# B&R Automation Studio project PLC code - cp (part 7)

#### BRSE_MB_Config.c
```c
/*! \file BRSE_MB_Config.c */

#include "BRSE_MB_Main.h"

BRSE_MB_ServerCfg_typ gBRSE_MB_Internal;

/*! \interface BRSE_MB_Alloc
	\brief Server: Function for allocating a modbus server unit.

	\param[in] 	Unit	Identity of the unit (0-255)
	\param[in]	MaxCoils	The maximum number of coils (references) used in this unit.
	\param[in]	MaxHoldingRegisters	The maximum number of holding registers used in this unit.
	\param[in] MaxDiscreteInputs	The maximum number of discrete inputs used in this unit.
	\param[in] MaxInputRegisters	The maximum number of input registers used in this unit.
	\param[out] Returns a pointer to the internal structure. Can be used for debug purposes.

*/
unsigned long BRSE_MB_Alloc(unsigned char Unit, unsigned short MaxCoils, unsigned short MaxHoldingRegisters, unsigned short MaxDiscreteInputs, unsigned short MaxInputRegisters)
{
	UINT status = 0;
	if (gBRSE_MB_Internal.Unit[Unit].pCoils || gBRSE_MB_Internal.Unit[Unit].pDiscreteInputs ||
		gBRSE_MB_Internal.Unit[Unit].pInputRegisters || gBRSE_MB_Internal.Unit[Unit].pHoldingRegisters)
		return BRSE_MB_ERR_UNIT_ALLOCATED; /* Unit can only be allocated once */

	memset(&gBRSE_MB_Internal.Unit[Unit], 0, sizeof(gBRSE_MB_Internal.Unit[Unit]));
	gBRSE_MB_Internal.Unit[Unit].MaxCoils = MaxCoils;
	gBRSE_MB_Internal.Unit[Unit].MaxDiscreteInputs = MaxDiscreteInputs;
	gBRSE_MB_Internal.Unit[Unit].MaxHoldingRegisters = MaxHoldingRegisters;
	gBRSE_MB_Internal.Unit[Unit].MaxInputRegisters = MaxInputRegisters;

	if (MaxCoils > 0)
	{
		status = TMP_alloc(MaxCoils*sizeof(UDINT) , (void **)&(gBRSE_MB_Internal.Unit[Unit].pCoils));
		if (status == 0)
			memset((void *)gBRSE_MB_Internal.Unit[Unit].pCoils, 0, MaxCoils*sizeof(UDINT));
		else
			ERRxwarning(status,(UDINT)gBRSE_MB_Internal.Unit[Unit].pCoils,(void *)"Coils: No memory!");
	}

	if (status != 0) /* reset unit */
	{
		memset(&gBRSE_MB_Internal.Unit[Unit], 0, sizeof(gBRSE_MB_Internal.Unit[Unit]));
		return status;
	}

	if (MaxDiscreteInputs > 0)
	{
		status = TMP_alloc(MaxDiscreteInputs*sizeof(UDINT) , (void **)&(gBRSE_MB_Internal.Unit[Unit].pDiscreteInputs));
		if (status == 0)
			memset((void *)gBRSE_MB_Internal.Unit[Unit].pDiscreteInputs, 0, MaxDiscreteInputs*sizeof(UDINT));
		else
			ERRxwarning(status,(UDINT)gBRSE_MB_Internal.Unit[Unit].pDiscreteInputs,(void *)"DiscreteI: No memory!");
	}

	if (status != 0) /* reset unit */
	{
		memset(&gBRSE_MB_Internal.Unit[Unit], 0, sizeof(gBRSE_MB_Internal.Unit[Unit]));
		return status;
	}

	if (MaxHoldingRegisters > 0)
	{
		status = TMP_alloc(MaxHoldingRegisters*sizeof(UDINT) , (void **)&(gBRSE_MB_Internal.Unit[Unit].pHoldingRegisters));
		if (status == 0)
			memset((void *)gBRSE_MB_Internal.Unit[Unit].pHoldingRegisters, 0, MaxHoldingRegisters*sizeof(UDINT));
		else
			ERRxwarning(status,(UDINT)gBRSE_MB_Internal.Unit[Unit].pHoldingRegisters,(void *)"HoldingR: No memory!");
	}

	if (status != 0) /* reset unit */
	{
		memset(&gBRSE_MB_Internal.Unit[Unit], 0, sizeof(gBRSE_MB_Internal.Unit[Unit]));
		return status;
	}

	if (MaxInputRegisters > 0)
	{
		status = TMP_alloc(MaxInputRegisters*sizeof(UDINT) , (void **)&(gBRSE_MB_Internal.Unit[Unit].pInputRegisters));
		if (status == 0)
			memset((void *)gBRSE_MB_Internal.Unit[Unit].pInputRegisters, 0, MaxInputRegisters*sizeof(UDINT));
		else
			ERRxwarning(status,(UDINT)gBRSE_MB_Internal.Unit[Unit].pInputRegisters,(void *)"InputReg:  No memory!");
	}

	if (status != 0) /* reset unit */
	{
		memset(&gBRSE_MB_Internal.Unit[Unit], 0, sizeof(gBRSE_MB_Internal.Unit[Unit]));
	}

	return (unsigned long)&gBRSE_MB_Internal;
}

/*! \interface BRSE_MB_Coil
	\brief Server: Function binding a coil to a variable

	Note that this function uses relative modbus adressing. Reference 0 corresponds to Modbus adress 1.

	\param[in] 	Unit	Identity of the unit (0-255)
	\param[in]	Reference	Coil address within unit (0..MaxCoils-1 in Alloc)
	\param[in]	VariableAddress	Address of the boolean variable.
	\param[out] Returns 0 or an error code.
*/
unsigned short BRSE_MB_Coil(unsigned char Unit, unsigned short Reference, unsigned long PvAddress)
{
	UDINT *coils;
	if (Reference >= gBRSE_MB_Internal.Unit[Unit].MaxCoils || PvAddress == 0)
		return BRSE_MB_ERR_REFERENCE;
	coils = (UDINT *)gBRSE_MB_Internal.Unit[Unit].pCoils; /* use as dynamic UDINT[] */
	coils[Reference] = PvAddress;
	return 0;
}

/*! \interface BRSE_MB_HoldingRegister
	\brief Server: Function binding a holding register to a variable

	Note that this function uses relative modbus adressing. Reference 0 corresponds to Modbus adress 40001.

	\param[in] 	Unit	Identity of the unit (0-255)
	\param[in]	Reference	Holding register address within unit (0..MaxHoldingRegisters-1 in Alloc)
	\param[in]	VariableAddress	Address of the integer variable.
	\param[out] Returns 0 or an error code.
*/
unsigned short BRSE_MB_HoldingRegister(unsigned char Unit, unsigned short Reference, unsigned long PvAddress)
{
	UDINT *holdingRegisters;
	if (Reference >= gBRSE_MB_Internal.Unit[Unit].MaxHoldingRegisters || PvAddress == 0)
		return BRSE_MB_ERR_REFERENCE;
	holdingRegisters = (UDINT *)gBRSE_MB_Internal.Unit[Unit].pHoldingRegisters; /* use as dynamic UDINT[] */
	holdingRegisters[Reference] = PvAddress;
	return 0;
}

/*! \interface BRSE_MB_4ByteHoldingRegister
	\brief Server: Function binding a 4 byte variable to 2 holding registers

	Note that this function uses relative modbus adressing. Reference 0 corresponds to Modbus adress 40001.

	\param[in] 	Unit	Identity of the unit (0-255)
	\param[in]	Reference	Holding register address within unit (0..MaxHoldingRegisters-1 in Alloc). Next free modbus address will be Reference+2 as the function assumes that you bind a 4-byte variable.
	\param[in]	VariableAddress	Address of the 4 byte variable.
	\param[out] Returns 0 or an error code.
*/
unsigned short BRSE_MB_4ByteHoldingRegister(unsigned char Unit, unsigned short Reference, unsigned long PvAddress)
{
	UDINT *holdingRegisters;
	if (Reference + 1 >= gBRSE_MB_Internal.Unit[Unit].MaxHoldingRegisters || PvAddress == 0)
		return BRSE_MB_ERR_REFERENCE;
	holdingRegisters = (UDINT *)gBRSE_MB_Internal.Unit[Unit].pHoldingRegisters; /* use as dynamic UDINT[] */
	holdingRegisters[Reference] = 1;
	holdingRegisters[Reference + 1] = PvAddress;
	return 0;
}
/*! \interface BRSE_MB_InputRegister
	\brief Server: Function binding a input register to a variable

	Note that this function uses relative modbus adressing. Reference 0 corresponds to Modbus adress 30001

	\param[in] 	Unit	Identity of the unit (0-255)
	\param[in]	Reference	Input register address within unit (0..MaxInputRegister-1 in Alloc)
	\param[in]	VariableAddress	Address of the integer variable.
	\param[out] Returns 0 or an error code.
*/
unsigned short BRSE_MB_InputRegister(unsigned char Unit, unsigned short Reference, unsigned long PvAddress)
{
	UDINT *inputRegisters;
	if (Reference >= gBRSE_MB_Internal.Unit[Unit].MaxInputRegisters || PvAddress == 0)
		return BRSE_MB_ERR_REFERENCE;
	inputRegisters = (UDINT *)gBRSE_MB_Internal.Unit[Unit].pInputRegisters; /* use as dynamic UDINT[] */
	inputRegisters[Reference] = PvAddress;
	return 0;
}

/*! \interface BRSE_MB_DiscreteInput
	\brief Server: Function binding a coil to a variable

	Note that this function uses relative modbus adressing. Reference 0 corresponds to Modbus adress 10001.

	\param[in] 	Unit	Identity of the unit (0-255)
	\param[in]	Reference	Coil address within unit (0..MaxDiscreteInputs-1 in Alloc)
	\param[in]	VariableAddress	Address of the boolean variable.
	\param[out] Returns 0 or an error code.
*/
unsigned short BRSE_MB_DiscreteInput(unsigned char Unit, unsigned short Reference, unsigned long PvAddress)
{
	UDINT *discreteInputs;
	if (Reference >= gBRSE_MB_Internal.Unit[Unit].MaxDiscreteInputs || PvAddress == 0)
		return BRSE_MB_ERR_REFERENCE;
	discreteInputs = (UDINT *)gBRSE_MB_Internal.Unit[Unit].pDiscreteInputs; /* use as dynamic UDINT[] */
	discreteInputs[Reference] = PvAddress;
	return 0;
}
```

#### BRSE_MB_Server.c
```c
/*! \file BRSE_MB_Server.c */

#include <bur/plctypes.h>
#include "BRSE_MB.h"
#include "BRSE_MB_Main.h"

/***************************/
/* Necessary byte swapping */
/***************************/
#ifdef _SG4
	#define SWAPUINT	swapUINT
	#define SWAPINT		swapINT
#else
	#define SWAPUINT
	#define SWAPINT
#endif

extern BRSE_MB_ServerCfg_typ gBRSE_MB_Internal; /* declared in BRSE_MB_Config.c */

 /*!
	\interface BRSE_MB_Server
	\brief Server: Interprets a byte buffer and creates a response to it according to modbus specification.
	Units and variables are configured with other BRSE_MB-functions.

	\param[in] Unit			The unit identifier (0-254)
	\param[in]	ClientFormat	Set the format of 4 byte variables to Intel or Motorola. BRSE_MB_INTEL / BRSE_MB_MOTOROLA

	\param[in] InputBuffer	The modbus byte buffer to respond to.
		Byte 0 is the function code.
		Byte 1-2 is the reference number (offset within unit where to start reading/writing).

	\param[out] OutputBuffer	The response buffer
	\param[out] BufferLength	The total number of bytes in the output buffer
	\param[out] Status			Return status.

*/
void BRSE_MB_Server(struct BRSE_MB_Server* inst)
{
	UINT	uintVar;
	/*****************************************/
	/* Check inputs and reset function block */
	/*****************************************/
	if (
		 (	!gBRSE_MB_Internal.Unit[inst->Unit].pCoils && !gBRSE_MB_Internal.Unit[inst->Unit].pDiscreteInputs &&
			!gBRSE_MB_Internal.Unit[inst->Unit].pInputRegisters && !gBRSE_MB_Internal.Unit[inst->Unit].pHoldingRegisters)
		)/* Unit not allocated */
	{
		inst->Status = BRSE_MB_ERR_ILLEGAL_FUNCTION; /* Unit is unconfigured and cannot process any request */
		return;
	}

	memset(&inst->OutputBuffer, 0, sizeof(inst->OutputBuffer));
	memset(&inst->Request, 0, sizeof(inst->Request));

	/*****************************/
	/* Parse request information */
	/*****************************/

	/* Function code (byte 0) */
	inst->Request.Type = inst->InputBuffer[0];
	if (inst->Request.Type == 0) /* FC 0 does not exist */
	{
		inst->Status = BRSE_MB_ERR_ILLEGAL_FUNCTION;
		return;
	}
	/* Reference number (byte 1,2) */
	memcpy(&uintVar, &inst->InputBuffer[1], sizeof(uintVar));
	inst->Request.StartAddr = SWAPUINT(uintVar);

	if(inst->Request.Type == BRSE_MB_WRITE_SINGLE_COIL || inst->Request.Type == BRSE_MB_WRITE_SINGLE_REGISTER)
	{
		inst->Request.Quantity = 1;
	}
	else /* Word/bit count (byte 3,4) */
	{
		memcpy(&uintVar, &inst->InputBuffer[3], sizeof(uintVar));
		inst->Request.Quantity = SWAPUINT(uintVar);
	}
	if (inst->Request.Quantity == 0)
	{
		inst->Status = BRSE_MB_ERR_ILLEGAL_DATA_ADDRESS;
		return;
	}

	/**************************************/
	/* Analyze request and build response */
	/**************************************/
	inst->OutputBuffer[0] = inst->Request.Type; /* Echo function code */

	switch(inst->Request.Type)
	{
		case BRSE_MB_READ_COILS:					/* 0x01 */
			inst->Status = BRSE_MB_ReadCoils(inst);
			break;

		case BRSE_MB_READ_DISCRETE_INPUTS:			/* 0x02 */
			inst->Status = BRSE_MB_ReadDiscreteInputs(inst);
			break;

		case BRSE_MB_READ_HOLDING_REGISTERS:		/* 0x03 */
			inst->Status = BRSE_MB_ReadHoldingRegisters(inst);
			break;

		case BRSE_MB_READ_INPUT_REGISTERS:			/* 0x04 */
			inst->Status = BRSE_MB_ReadInputRegisters(inst);
			break;

		case BRSE_MB_WRITE_SINGLE_COIL:				/* 0x05 */
			inst->Status = BRSE_MB_WriteSingleCoil(inst);
			break;

		case BRSE_MB_WRITE_SINGLE_REGISTER:			/* 0x06 */
			inst->Status = BRSE_MB_WriteSingleRegister(inst);
			break;

		case BRSE_MB_WRITE_MULTIPLE_COILS:			/* 0x0F */
			inst->Status = BRSE_MB_WriteMultipleCoils(inst);
			break;

		case BRSE_MB_WRITE_MULTIPLE_REGISTERS:		/* 0x10 */
			inst->Status = BRSE_MB_WriteMultipleRegisters(inst);
			break;

		default:
			inst->Status = BRSE_MB_ERR_ILLEGAL_FUNCTION;
			break;
	}
	if (inst->Status != 0) /* Reset outputs */
		memset(&inst->OutputBuffer, 0, sizeof(inst->OutputBuffer));

}

UINT BRSE_MB_ReadCoils(struct BRSE_MB_Server* inst)
{
	UDINT 				*coils;
	if(inst->Request.StartAddr + inst->Request.Quantity <= gBRSE_MB_Internal.Unit[inst->Unit].MaxCoils
		&& inst->Request.Quantity <= BRSE_MB_MAX_COILS
		&& gBRSE_MB_Internal.Unit[inst->Unit].pCoils)
	{
		coils = (UDINT *)gBRSE_MB_Internal.Unit[inst->Unit].pCoils; /* use as dynamic UDINT[] */
		return BRSE_MB_FillDigitalBuffer(inst, coils);
	}
	else
	{
		return BRSE_MB_ERR_ILLEGAL_DATA_ADDRESS;
	}
}

UINT BRSE_MB_ReadDiscreteInputs(struct BRSE_MB_Server* inst)
{
	UDINT 				*discreteInputs;
	if(inst->Request.StartAddr + inst->Request.Quantity <= gBRSE_MB_Internal.Unit[inst->Unit].MaxDiscreteInputs
		&& inst->Request.Quantity <= BRSE_MB_MAX_DISCRETE_INPUTS
		&& gBRSE_MB_Internal.Unit[inst->Unit].pDiscreteInputs)
	{
		discreteInputs = (UDINT *)gBRSE_MB_Internal.Unit[inst->Unit].pDiscreteInputs; /* use as dynamic UDINT[] */
		return BRSE_MB_FillDigitalBuffer(inst, discreteInputs);
	}
	else
	{
		return BRSE_MB_ERR_ILLEGAL_DATA_ADDRESS;
	}
}

UINT BRSE_MB_ReadHoldingRegisters(struct BRSE_MB_Server* inst)
{
	UDINT *holdingRegisters;
	if (inst->Request.StartAddr + inst->Request.Quantity <= gBRSE_MB_Internal.Unit[inst->Unit].MaxHoldingRegisters
		&& inst->Request.Quantity <= BRSE_MB_MAX_HOLDING_REG_READ
		&& gBRSE_MB_Internal.Unit[inst->Unit].pHoldingRegisters)
	{
		holdingRegisters = (UDINT *)gBRSE_MB_Internal.Unit[inst->Unit].pHoldingRegisters; /* use as dynamic UDINT[] */
		return BRSE_MB_FillRegisterBuffer(inst, holdingRegisters);
	}
	else
	{
		return BRSE_MB_ERR_ILLEGAL_DATA_ADDRESS;
	}
}

UINT BRSE_MB_ReadInputRegisters(struct BRSE_MB_Server* inst)
{
	UDINT *inputRegisters;
	if (inst->Request.StartAddr + inst->Request.Quantity <= gBRSE_MB_Internal.Unit[inst->Unit].MaxInputRegisters
		&& inst->Request.Quantity <= BRSE_MB_MAX_INPUT_REG_READ
		&& gBRSE_MB_Internal.Unit[inst->Unit].pInputRegisters)
	{
		inputRegisters = (UDINT *)gBRSE_MB_Internal.Unit[inst->Unit].pInputRegisters; /* use as dynamic UDINT[] */
		return BRSE_MB_FillRegisterBuffer(inst, inputRegisters);
	}
	else
	{
		return BRSE_MB_ERR_ILLEGAL_DATA_ADDRESS;
	}
}

/*
 Response looks like
   Byte
	0:			FC
	1-2:		Reference
	3:			FF=0N, 00=OFF
	4:			0

	sets BufferLength = 5
 */
UINT BRSE_MB_WriteSingleCoil(struct BRSE_MB_Server* inst)
{
	UINT uintVar;
	UINT value;
	UDINT *coils;

	inst->BufferLength = 5;
	if(inst->Request.StartAddr < gBRSE_MB_Internal.Unit[inst->Unit].MaxCoils && gBRSE_MB_Internal.Unit[inst->Unit].pCoils)
	{
		coils = (UDINT *)gBRSE_MB_Internal.Unit[inst->Unit].pCoils; /* use as dynamic UDINT[] */
		memcpy(&uintVar, &inst->InputBuffer[3], sizeof(uintVar)); /* value */
		value = SWAPUINT(uintVar);

		memcpy(&inst->OutputBuffer[1], &inst->InputBuffer[1], 2); /* Reference: 2 byte */
		memcpy(&inst->OutputBuffer[3], &inst->InputBuffer[3], 2); /* Value: 2 byte */

		if (coils[inst->Request.StartAddr])
		{
			if(value == BRSE_MB_ON)
				*((BOOL*)(coils[inst->Request.StartAddr])) = 1;
			else
				*((BOOL*)(coils[inst->Request.StartAddr])) = 0;
		}
	}
	else
	{
		return BRSE_MB_ERR_ILLEGAL_DATA_ADDRESS;
	}
	return 0;
}

/*
 Response looks like
   Byte
	0:			FC
	1-2:		Reference
	3-4:		Register value

	sets BufferLength = 5
 */
UINT BRSE_MB_WriteSingleRegister(struct BRSE_MB_Server* inst)
{
	INT intVar;
	INT value;
	UDINT *holdingRegisters;

	inst->BufferLength = 5;

	if(inst->Request.StartAddr < gBRSE_MB_Internal.Unit[inst->Unit].MaxHoldingRegisters && gBRSE_MB_Internal.Unit[inst->Unit].pHoldingRegisters)
	{
		holdingRegisters = (UDINT *)gBRSE_MB_Internal.Unit[inst->Unit].pHoldingRegisters; /* use as dynamic UDINT[] */
		memcpy(&intVar, &(inst->InputBuffer[3]), sizeof(intVar)); /* value */
		value = SWAPUINT(intVar);

		memcpy(&inst->OutputBuffer[1], &inst->InputBuffer[1], 2); /* Reference: 2 byte */
		memcpy(&inst->OutputBuffer[3], &inst->InputBuffer[3], 2); /* Value: 2 byte */

		if (holdingRegisters[inst->Request.StartAddr] > 1) /*check that its not a 4-byte holding!*/
			*((INT*)(holdingRegisters[inst->Request.StartAddr])) = value;
		else
			return BRSE_MB_ERR_ILLEGAL_DATA_ADDRESS;
	}
	else
	{
		return BRSE_MB_ERR_ILLEGAL_DATA_ADDRESS;
	}

	return 0;
}

/*
 Response looks like
   Byte
	0:			FC
	1-2:		Reference
	3-4:		Bit count

	sets BufferLength = 5
 */
UINT BRSE_MB_WriteMultipleCoils(struct BRSE_MB_Server* inst)
{
	UINT i;
	UDINT *coils;

	inst->BufferLength = 5;
	if(inst->Request.StartAddr + inst->Request.Quantity <= gBRSE_MB_Internal.Unit[inst->Unit].MaxCoils
		&& inst->Request.Quantity <= BRSE_MB_MAX_COILS_WRITE
		&& gBRSE_MB_Internal.Unit[inst->Unit].pCoils)
	{
		coils = (UDINT *)gBRSE_MB_Internal.Unit[inst->Unit].pCoils; /* use as dynamic UDINT[] */
		memcpy(&inst->OutputBuffer[1], &inst->InputBuffer[1], 2);		/* Reference: 2 byte */
		memcpy(&inst->OutputBuffer[3], &inst->InputBuffer[3], 2);  	/* Bit count: 2 byte */

		for(i=0; i < inst->Request.Quantity; i++)
		{
			if (coils[inst->Request.StartAddr+i])
			{
				if ((inst->InputBuffer[6 + (i/8)] & (USINT)(0x01 << (i%8))) && (coils[inst->Request.StartAddr+i]))
					*((BOOL*)(coils[inst->Request.StartAddr+i])) = 1;
				else
					*((BOOL*)(coils[inst->Request.StartAddr+i])) = 0;
			}
		}
		return 0;
	}
	else
	{
		return BRSE_MB_ERR_ILLEGAL_DATA_ADDRESS;
	}

}
/*
 Response looks like
   Byte
	0:			FC
	1-2:		Reference
	3-4:		Word count

	sets BufferLength = 5
 */
UINT BRSE_MB_WriteMultipleRegisters(struct BRSE_MB_Server* inst)
{
	INT							int_var1, int_var2;
	UINT						i;
	UDINT *holdingRegisters;

	inst->BufferLength = 5;

	if (inst->Request.StartAddr + inst->Request.Quantity <= gBRSE_MB_Internal.Unit[inst->Unit].MaxHoldingRegisters
		&& inst->Request.Quantity <= BRSE_MB_MAX_HOLDING_REG_WRITE
		&& gBRSE_MB_Internal.Unit[inst->Unit].pHoldingRegisters)
	{

			holdingRegisters = (UDINT *)gBRSE_MB_Internal.Unit[inst->Unit].pHoldingRegisters; /* use as dynamic UDINT[] */
			memcpy(&inst->OutputBuffer[1], &inst->InputBuffer[1], 2);	/* 	Reference: 2 byte */
			memcpy(&inst->OutputBuffer[3], &inst->InputBuffer[3], 2); 	/* Value: 2 byte */

			for(i=0; i < inst->Request.Quantity; i++)
			{
				if (holdingRegisters[inst->Request.StartAddr+i] == 0)
				{
					return BRSE_MB_ERR_ILLEGAL_DATA_ADDRESS;
				}

				if (holdingRegisters[inst->Request.StartAddr+i] == 1 && holdingRegisters[inst->Request.StartAddr+i+1]) /* 4 byte variable */
				{
					memcpy(&int_var1, &inst->InputBuffer[6+(i*2)], sizeof(int_var1));
					memcpy(&int_var2, &inst->InputBuffer[6+(i*2)+2], sizeof(int_var2));
					if (inst->ClientFormat == BRSE_MB_INTEL )
					{
						#ifdef _SG4
						*((INT*)(holdingRegisters[inst->Request.StartAddr+i+1])) = SWAPINT(int_var1);
						*((INT*)(holdingRegisters[inst->Request.StartAddr+i+1]+2)) = SWAPINT(int_var2);
						#else
						*((INT*)(holdingRegisters[inst->Request.StartAddr+i+1])) = SWAPINT(int_var2);
						*((INT*)(holdingRegisters[inst->Request.StartAddr+i+1]+2)) = SWAPINT(int_var1);
						#endif
					}
					else
					{
						#ifdef _SG4
						*((INT*)(holdingRegisters[inst->Request.StartAddr+i+1])) = SWAPINT(int_var2);
						*((INT*)(holdingRegisters[inst->Request.StartAddr+i+1]+2)) = SWAPINT(int_var1);
						#else
						*((INT*)(holdingRegisters[inst->Request.StartAddr+i+1])) = SWAPINT(int_var1);
						*((INT*)(holdingRegisters[inst->Request.StartAddr+i+1]+2)) = SWAPINT(int_var2);
						#endif
					}

					i++;
				}
				else if (holdingRegisters[inst->Request.StartAddr+i] > 1) /* Normal 2 byte register */
				{
					memcpy(&int_var1, &inst->InputBuffer[6+(i*2)], sizeof(int_var1));
					*((INT*)(holdingRegisters[inst->Request.StartAddr+i])) = SWAPINT(int_var1);
				}
			}

			return 0;
	}
	else
	{
		return BRSE_MB_ERR_ILLEGAL_DATA_ADDRESS;
	}
}

/*********************/
/* Utility functions */
/*********************/
/*
 Response looks like
   Byte
	0:			FC
	1:			Byte count of response (B=(bit count +7)/8)
	2-(B+1):	Bit values

	sets BufferLength = 2+B
 */
UINT BRSE_MB_FillDigitalBuffer(struct BRSE_MB_Server* inst, UDINT *boolPtrArray)
{
	UINT				i;
	USINT				byte_nr;
	/* Number of bytes in response (1) */
	if ((inst->Request.Quantity % 8) > 0)	byte_nr = (inst->Request.Quantity / 8) + 1;
	else									byte_nr = (inst->Request.Quantity / 8);
	inst->OutputBuffer[1] = byte_nr;

	/* Value of boolean boolPtrArray (2->byte_nr) */
	for(i = 0; i < inst->Request.Quantity; i++)
	{
		/* if pv assigned and true */
		if( boolPtrArray[inst->Request.StartAddr+i] && (*((BOOL *)boolPtrArray[inst->Request.StartAddr+i])))
			inst->OutputBuffer[2 + (i/8)] = inst->OutputBuffer[2 + (i/8)] | (USINT)(0x01 << (i%8));
		else
			inst->OutputBuffer[2 + (i/8)] = inst->OutputBuffer[2 + (i/8)] & (USINT)~(0x01 << (i%8));

	}
	inst->BufferLength = 2+byte_nr;
	return 0;
}

/*
 Response looks like
   Byte
	0:			FC
	1:			Byte count of response (B=2*word count)
	2-(B+1):	Register values (1-125)

	returns BufferLength = 2+2*(word count)
 */
UINT BRSE_MB_FillRegisterBuffer(struct BRSE_MB_Server* inst, UDINT *intPtrArray)
{
	INT				int_var1, int_var2;
	UINT			i;

	inst->OutputBuffer[1] = inst->Request.Quantity * 2; /* nbr data bytes */

	for(i = 0; i < inst->Request.Quantity; i++)
	{
		if(intPtrArray[inst->Request.StartAddr + i])
		{
			if(intPtrArray[inst->Request.StartAddr + i] == 1 && intPtrArray[inst->Request.StartAddr + i + 1]) /*4-byte*/
			{
				int_var1 = SWAPINT(*((INT*)(intPtrArray[inst->Request.StartAddr + i + 1])));
				int_var2 = SWAPINT(*((INT*)(intPtrArray[inst->Request.StartAddr + i + 1]+2)));

				if(inst->ClientFormat == BRSE_MB_INTEL)
				{
					#ifdef _SG4
						memcpy(&inst->OutputBuffer[2 + (i*2)], &int_var1, sizeof(int_var1));
						memcpy(&inst->OutputBuffer[2 + ((i+1)*2)], &int_var2, sizeof(int_var2));
					#else
						memcpy(&inst->OutputBuffer[2 + (i*2)], &int_var2, sizeof(int_var2));
						memcpy(&inst->OutputBuffer[2 + ((i+1)*2)], &int_var1, sizeof(int_var1));
					#endif
				}
				else
				{
					#ifdef _SG4
						memcpy(&inst->OutputBuffer[2 + (i*2)], &int_var2, sizeof(int_var2));
						memcpy(&inst->OutputBuffer[2 + ((i+1)*2)], &int_var1, sizeof(int_var1));
					#else
						memcpy(&inst->OutputBuffer[2 + (i*2)], &int_var1, sizeof(int_var1));
						memcpy(&inst->OutputBuffer[2 + ((i+1)*2)], &int_var2, sizeof(int_var2));
					#endif
				}

				i++;
			}
			else if(intPtrArray[inst->Request.StartAddr + i] > 1) /*just in case, normally it shouldnt be 1 here anyhow*/
			{
				int_var1 = SWAPINT(*((INT*)(intPtrArray[inst->Request.StartAddr + i])));
				memcpy(&inst->OutputBuffer[2 + (i*2)], &int_var1, sizeof(int_var1));
			}
		}
		else /*bad pointer*/
		{
			int_var1 = 0;
			memcpy(&inst->OutputBuffer[2 + (i*2)], &int_var1, sizeof(int_var1));
		}
	}
	inst->BufferLength = 2+2*inst->Request.Quantity;
	return 0;
}
```

#### MB_RequestQueue.c
```c
/*! \file MB_RequestQueue.c */

#include <bur/plctypes.h>
#include "BRSE_MB.h"
#include "BRSE_MB_Main.h"

#define	BUSY				65535

extern MB_ClientStruct_typ gMB_ClientInternal;

UINT MB_AckClientRequest(USINT ClientID, UINT ReturnStatus)
{
	MB_Client_typ *pQueue;
	MB_ClientQueueItem_typ *pQueueItem;
	UINT status = 0;

	if (gMB_ClientInternal.pClients[ClientID] == 0)
		return MB_ERR_CLIENT_NOT_ALLOCATED;

	pQueue = (MB_Client_typ *)gMB_ClientInternal.pClients[ClientID];
	if ((*pQueue).Lock)
	{
		status = BUSY;
		return status;
	}

	/* -- Begin synchronized block -- */
	(*pQueue).Lock = 1; /* prevent others from reading from / writing to queue */
	pQueueItem = &((*pQueue).Queue[(*pQueue).IndexExec]);
	(*((UINT *) ((*pQueueItem).StatusAddr))) = ReturnStatus;
	(*pQueue).IndexExec++;
	(*pQueue).IndexExec %= (MB_QUEUE_SIZE+1);
	memset(pQueueItem, 0, sizeof(*pQueueItem));
	(*pQueue).Lock = 0;
	/* -- End synchronized block -- */
	return status;
}

UINT MB_AddToRequestQueue(USINT clientID, USINT fc, UINT quantity, UINT startAddress, UDINT variableAddress, UDINT statusAddress, USINT Unit)
{
	MB_Client_typ *pQueue;
	MB_ClientQueueItem_typ *pQueueItem;
	UINT status = 0;

	if (gMB_ClientInternal.pClients[clientID] == 0)
		return MB_ERR_CLIENT_NOT_ALLOCATED;

	pQueue = (MB_Client_typ *)gMB_ClientInternal.pClients[clientID];
	if ((*pQueue).Lock)
	{
		status = BUSY;
		return status;
	}

	/* -- Begin synchronized block -- */
	(*pQueue).Lock = 1; /* prevent others from reading from / writing to queue */
	pQueueItem = &((*pQueue).Queue[(*pQueue).IndexInsert]);
	if (((*pQueue).IndexExec == (*pQueue).IndexInsert) && ((*pQueueItem).VariableAddr != 0))
	{
		status = MB_ERR_QUEUE_FULL;
	}
	else
	{
		(*((UINT *)statusAddress)) = BUSY;
		(*pQueueItem).Request.Unit = Unit;
		(*pQueueItem).Request.Quantity = quantity;
		(*pQueueItem).Request.Type = fc;
		(*pQueueItem).Request.StartAddr = startAddress;
		(*pQueueItem).VariableAddr = variableAddress;
		(*pQueueItem).StatusAddr = statusAddress;
		(*pQueue).IndexInsert++;
		(*pQueue).IndexInsert %= (MB_QUEUE_SIZE+1);
	}
	(*pQueue).Lock = 0;
	/* -- End synchronized block -- */
	return status;
}

USINT MB_QueueStatus(USINT ClientID)
{
	MB_Client_typ *pQueue;
	USINT status = 0;

	if (gMB_ClientInternal.pClients[ClientID] == 0)
		return 0;

	pQueue = (MB_Client_typ *)gMB_ClientInternal.pClients[ClientID];
	if ((*pQueue).Lock)
	{
		return 1;
	}
	/* Synchronized block */
	(*pQueue).Lock = 1;
	if ((*pQueue).IndexExec == (*pQueue).IndexInsert) /* queue empty */
		status = 0;
	else
		status = 1;
	(*pQueue).Lock = 0;
	/* Synchronized end */
	return status;
}
```

### Library Logical/ExtPack/_Comms/ModbusComms/ModbusComms_v1/Libraries/BRSE_MBT

#### BRSE_MBT.var
```iecst
VAR CONSTANT
	BRSE_MBT_MAX_BUFFER : UINT := 261;
	BRSE_MBT_MAX_CLIENT : USINT := 20;
	BRSE_MBT_ERR_TOO_MANY_CLIENTS : UINT := 30001;
	BRSE_MBT_LOG_MAX : UINT := 50;
	MBT_RECEIVE_TIMEOUT : UDINT := 3000; (*Await response timeout, ms (cycle time=0 --> never timeout)*)
	BRSE_MBT_RESEND_LIMIT : UINT := 5; (*Number of times to resend before trying to re-establish connection*)
	BRSE_MBT_RETRY_PERIOD : UINT := 10000; (*If error occurs on TcpOpen or TcpClient, wait this time before retrying. (cycle time assumed 10ms if set to 0)*)
	BRSE_DISCONNECT_TIMEOUT : TIME := T#60S; (*Disconnects clients after this time without activity*)
END_VAR
```

#### BRSE_MBT.fun
```iecst
FUNCTION_BLOCK BRSE_MBT_Server
	VAR_INPUT
		Enable : BOOL; (*Add your parameter comment*)
		ClientFormat : USINT;
		Port : UINT;
		SocketTimeout : UDINT; (*Linger time for incoming sockets*)
	END_VAR
	VAR_OUTPUT
		Status : UINT;
	END_VAR
	VAR
		FB_TcpOpen : TcpOpen;
		FB_TcpServer : TcpServer;
		FB_TcpCloseOld : TcpClose;
		FB_TcpCloseServer : TcpClose;
		FB_TcpClose : ARRAY[0..BRSE_MBT_MAX_CLIENT] OF TcpClose;
		Clients : ARRAY[0..BRSE_MBT_MAX_CLIENT] OF BRSE_MBT_Client_typ;
		Step : UINT;
		ClientNr : USINT;
		FB_BRSE_MB_Server : BRSE_MB_Server;
		Log : ARRAY[0..BRSE_MBT_LOG_MAX] OF STRING[100];
		LogIndex : UINT;
		TmpUINT : UINT;
		NewClient : BRSE_MBT_NewClient_typ;
		Error : UINT; (*Indicator to leave state when all fubs are done*)
		IsBusy : UINT; (*Indicates that one or more fubs are not ready to leave state*)
		TmpStr : STRING[10];
		LingerOptions : tcpLINGER_typ;
	END_VAR
END_FUNCTION_BLOCK

FUNCTION MBT_GetServerInternalStructAddr : UDINT (*Returns the allocated server struct address, i.e. a pointer to a BRSE_MBT_Internal_typ. Used only for debug purposes.*)
END_FUNCTION

FUNCTION MBT_GetClientInternalStructAddr : UDINT (*Returns the allocated client internal struct address, i.e. a pointer to a MBT_ClientInternal_typ. Used only for debug purposes.*)
END_FUNCTION

FUNCTION_BLOCK MBT_ServerExit (*Closes any open tcp port.*)
	VAR_OUTPUT
		Status : UINT;
	END_VAR
	VAR
		FB_TcpClose : TcpClose;
	END_VAR
END_FUNCTION_BLOCK

FUNCTION_BLOCK MBT_Client
	VAR_INPUT
		Enable : BOOL;
		ServerFormat : USINT;
		ClientID : USINT;
		IpAddr : STRING[18];
		Port : UINT;
		ConnectionTimeout : UDINT; (*Time in ms the client waits for new requests (from queue) before closing down the socket connection*)
		SocketTimeout : UDINT; (*Linger time for outgoing sockets*)
	END_VAR
	VAR_OUTPUT
		Status : UINT;
	END_VAR
	VAR
		Step : UINT;
		FB_MB_CreateClientRequest : MB_CreateClientRequest;
		FB_MB_PutClientResponse : MB_PutClientResponse;
		FB_TcpOpen : TcpOpen;
		FB_TcpClient : TcpClient;
		FB_TcpSend : TcpSend;
		FB_TcpRecive : TcpRecv;
		FB_TcpClose : TcpClose;
		FB_RTInfo : RTInfo;
		FB_TcpIoctl : TcpIoctl;
		RecvLen : UINT;
		SendBuffer : ARRAY[0..BRSE_MBT_MAX_BUFFER] OF USINT;
		ReceiveBuffer : ARRAY[0..BRSE_MBT_MAX_BUFFER] OF USINT;
		TransactionId : UINT;
		Timeout : UDINT;
		RecvTransactionId : UINT;
		ErrorStatus : UINT;
		ResendCounter : UINT;
		CycleTimeMs : UDINT; (*Task cycle time in ms*)
		ElapsedTime : UDINT;
		LingerOptions : tcpLINGER_typ;
	END_VAR
END_FUNCTION_BLOCK

FUNCTION_BLOCK MBT_ExitClient (*Closes any open tcp port.*)
	VAR_INPUT
		ClientID : USINT; (*Add your parameter comment*)
	END_VAR
	VAR_OUTPUT
		Status : UINT;
	END_VAR
	VAR
		FB_TcpClose : TcpClose;
	END_VAR
END_FUNCTION_BLOCK
```

#### BRSE_MBT_Main.h
```c
/*! \file BRSE_MBT_Main.h */

/*!	\mainpage BRSE_MBT

	\section Introduction

	This library is used for setting up a modbus server and a modbus client.

	The Modbus data model has a simple structure that differentiates
	between four basic data types:

	\arg Discrete Inputs (BOOL Read-Only)
	\arg Coils (BOOL Read-Write)
	\arg Input Registers (INT Read-Only)
	\arg Holding Registers (INT Read-Write)

	(The expression "Input" is seen from the Client side).
	\anchor tasks
	\section Example_tasks Example tasks

	The source code to the example tasks can be found
	<a href="y:\Application\Libraries\BRSE_MBT\Documentation\MBT_example_tasks.zip">here</a>.

	\section Server

	The BRSE_MBT_Server function block acts as a modbus server. When enabled, it opens the tcp port 502 and starts
	listen for incoming modbus messages.

	Requests from each client are responded to in the same cycle.

	That brings the execution time to depend very much on the server load, i.e. frequency of client requests.

	Therefore, the program executing BRSE_MBT_Server needs to be put in a task class with high tolerance.

	It is recommended that the program is put in a fast (10-20ms), low priority task with high tolerance.

	\image html y:\Application\Libraries\BRSE_MBT\Documentation\BRSE_MBT_Server.jpg

	Units must be allocated with the BRSE_MB_Alloc function in the BRSE_MB library.

	MBT_ServerExit closes open tcp ports and should be called in the exit routine of the program.

	\section Client

	The MBT_Client is used together with the master/client functions of the BRSE_MB library.
	When a request (for example "Read 100 coils on unit 2 starting on address 5") has been placed in queue,
	this function block creates a modbus message, sends it to the server/slave and awaits a response.
	If no response is given, it resends the message after a certain time.

	\image html y:\Application\Libraries\BRSE_MBT\Documentation\BRSE_MBT_Client.jpg

	The client must be allocated with the MB_AllocClient function in the BRSE_MB library. A certain client ID
	is passed to the alloc function and the same ID is passed to the MBT_Client function.

	MBT_ExitClient closes open tcp ports and should be called in the exit routine of the program.

*/

/*! \page Error_Numbers Error Numbers
	\section Error_Numbers Error Numbers

	\b 0 	BRSE_MBT_INTEL: The server/client uses the Intel format

	\b 1 	BRSE_MBT_MOTOROLA: The server/client uses the Motorola format

	\b 30001 BRSE_MBT_ERR_TOO_MANY_CLIENTS: Too many clients.

*/
#ifndef _BRSE_MBT_MAIN_
#define _BRSE_MBT_MAIN_

#include <bur/plctypes.h>
#include "BRSE_MBT.h"
#include <string.h>

#endif

/* Common functions */
UINT BRSE_MBT_AddClient(struct BRSE_MBT_Server* inst);
void BRSE_MBT_RemoveClient(struct BRSE_MBT_Server* inst, UINT clientIdx);
UINT BRSE_MBT_AnalyzeReqFromClient(struct BRSE_MBT_Server* inst, UINT clientIdx);
UINT BRSE_MBT_CreateErrorMessage(struct BRSE_MBT_Server* inst, UINT errorCode, UINT clientIdx);
```

#### Example_Server.c
```c
/*!

 \page Example_server Example Server
 \section Example_server Example Server

 \par Description
	This program set up an TCP modbus server on the ethernet port of the system

 \par Example
  Example \ref tasks can be found here.

\par MBserv.var
\code
VAR
	FB_BRSE_MBT_Server : BRSE_MBT_Server := (0);
	FB_MBT_ServerExit : MBT_ServerExit := (0);
	discreteInput : ARRAY[0..9] OF BOOL := [9(FALSE)];
	coil : ARRAY[0..10] OF BOOL := [10(FALSE)];
	inputRegister : ARRAY[0..11] OF INT := [11(0)];
	holdingRegister : ARRAY[0..9] OF INT := [9(0)];
	realValue : ARRAY[0..5] OF REAL :=[5(0.0)];
	i : USINT := 0;
END_VAR
\endcode

\par MBserv.st
\code
PROGRAM _INIT

	(* Create a Modbus server with unit identity = 0, Coil = 10, HoldingRegister = 20, DiscreteInputs = 9, InputRegister = 11 *)
	BRSE_MB_Alloc(0,10,20,9,11);

	(* Bind the coils *)
	FOR i:=0 TO 10 DO
		BRSE_MB_Coil(0,i,ADR(coil[i]));
	END_FOR;
	(* Bind the discrete inputs *)
	FOR i:=0 TO 9 DO
		BRSE_MB_DiscreteInput(0,i,ADR(discreteInput[i]));
	END_FOR;
	(* Bind the holdning registers *)
	FOR i:=0 TO 9 DO
		BRSE_MB_HoldingRegister(0,i,ADR(holdingRegister[i]));
	END_FOR;
	(* Bind the input registers *)
	FOR i:=0 TO 11 DO
		BRSE_MB_InputRegister(0,i,ADR(inputRegister[i]));
	END_FOR;

	(* Bind 4 byte holdning registers to REAL values*)
	FOR i:=0 TO 5 DO
		BRSE_MB_4ByteHoldingRegister(0, 10 + i*2,ADR(realValue[i]));
	END_FOR;

END_PROGRAM

PROGRAM _CYCLIC

	(* Enable the server, use INTEL alignment (little endian) for real Values *)
	FB_BRSE_MBT_Server(Enable := 1, ClientFormat := BRSE_MB_INTEL);

END_PROGRAM

PROGRAM _EXIT

	(* Close the open tcp port *)
	FB_MBT_ServerExit();

END_PROGRAM

\endcode
*/

/*

 Example on how to use the BRSE_MBT Library as a modbus server in C

#include <bur/plctypes.h>

#ifdef _DEFAULT_INCLUDES
 #include <AsDefault.h>
#endif

void _INIT MBRTestINIT( void )
{
	UINT i;

	BRSE_MB_Alloc(1, NbrCoils, NbrHoldingRegisters, NbrDiscreteInputs, NbrInputRegisters);

	for (i=0; i<NbrCoils; i++)
	{
		BRSE_MB_Coil(1, i, (UDINT)&Coils[i]);
	}
	for (i=0; i<NbrHoldingRegisters; i++)
	{
		BRSE_MB_HoldingRegister(1, i, (UDINT)&HoldingRegisters[i]);
	}
	for (i=0; i<NbrDiscreteInputs; i++)
	{
		BRSE_MB_DiscreteInput(1, i, (UDINT)&DiscreteInputs[i]);
	}
	for (i=0; i<NbrInputRegisters; i++)
	{
		BRSE_MB_InputRegister(1, i, (UDINT)&InputRegisters[i]);
	}

	FB_BRSE_MBT_Server.Enable = 1;
}

void _CYCLIC MBRTestCYCLIC( void )
{
	BRSE_MBT_Server(&FB_BRSE_MBR_Server);
}

*/
```

#### MBT_Client.c
```c
/*! \file MBT_Client.c */

#include "BRSE_MBT.h"
#include "BRSE_MBT_Main.h"

#ifdef _SG4
	#define SWAPUINT	swapUINT
	#define SWAPINT		swapINT
#else
	#define SWAPUINT
	#define SWAPINT
#endif

#define	BUSY			65535
#define DISABLE		65534

MBT_ClientInternal_typ BRSE_MBT_ClientInternal;

UDINT MBT_GetClientInternalStructAddr()
{
	return (UDINT)&BRSE_MBT_ClientInternal;
}

/*!
	\interface MBT_Client
	\brief Client: Create a connection to a physical Ethernet Port and open port 502 and starts	send requests and listen to response according to internal queue.

	\param[in]	Enable	Enables execution of the function.
	\param[in]	ServerFormat	Set the format of 4 byte variables to Intel or Motorola. BRSE_MB_INTEL / BRSE_MB_MOTOROLA
	\param[in]	ClientID	Identity created in AllocClient.
	\param[in]	IpAddr	Ip address to the modbus server.
	\param[in]	Port	Port on the modbus server.
	\param[in]	ConnectionTimeout	This input specifies the time in milliseconds that the client waits for new requests before closing the connection. If the input is zero, the connection is left open to the server until next request.
	\param[in]	SocketTimeout	Time in seconds that the system keeps the socket alive after closing it. This can be used as the oposite station still has some data to send. If the input is zero, the socket is closed immediately.
	\param[out] Status	Return status.
*/
void MBT_Client(struct MBT_Client* inst)
{
	UINT uintSwapped;
	inst->Status = BUSY;
	switch(inst->Step)
	{
		case 0: /* init */
			inst->FB_TcpSend.enable = 1;
			inst->FB_TcpSend.pData = (UDINT)&(inst->SendBuffer[0]);
			inst->FB_TcpRecive.enable = 1;
			inst->FB_TcpRecive.pData = (UDINT)&(inst->ReceiveBuffer[0]);
			inst->FB_TcpRecive.datamax = sizeof(inst->ReceiveBuffer);
			inst->FB_TcpOpen.options = 0;
			inst->FB_TcpOpen.enable = 1;
			inst->FB_TcpOpen.port = 0;
			inst->FB_TcpClient.enable = 1;
			inst->FB_TcpClose.enable = 1;
			inst->FB_RTInfo.enable = 1;
			inst->FB_TcpIoctl.enable = 1;
			inst->ElapsedTime = 0;
			inst->Step = 1;

			/* beware: fall-through */

		case 1: /* Get cycle time */
			RTInfo(&inst->FB_RTInfo);
			if (inst->FB_RTInfo.status == 0)
			{
				inst->CycleTimeMs = inst->FB_RTInfo.cycle_time/1000; /* Convert to millis from micros */
				inst->Step = 10;
			}
			else if (inst->FB_RTInfo.status != ERR_FUB_BUSY)
			{
				inst->Status = inst->FB_RTInfo.status;
				break;
			}
			/* beware: fall-through */

		case 10: /* enable/disable */
			inst->ErrorStatus = 0;
			if (inst->Enable)
				inst->Step = 20;
			else
				break;
			/* beware: fall-through if enabled */

		case 20: /* Get request from queue */
			memset(&(inst->SendBuffer[0]), 0, sizeof(inst->SendBuffer));
			memset(&(inst->ReceiveBuffer[0]), 0, sizeof(inst->ReceiveBuffer));
			inst->ElapsedTime = 0;
			inst->ResendCounter = 0;
			inst->Step = 21;
			/* beware: fall-through */

		case 21:
			inst->ElapsedTime += inst->CycleTimeMs;
			inst->FB_MB_CreateClientRequest.AdrByteBuffer = (UDINT)&inst->SendBuffer[7];
			inst->FB_MB_CreateClientRequest.ByteBufferLen = BRSE_MBT_MAX_BUFFER-7;
			inst->FB_MB_CreateClientRequest.ClientID = inst->ClientID;
			inst->FB_MB_CreateClientRequest.ServerFormat = inst->ServerFormat;
			MB_CreateClientRequest(&inst->FB_MB_CreateClientRequest);
			if (inst->FB_MB_CreateClientRequest.Status == 0 && inst->FB_MB_CreateClientRequest.RequestBufferLen > 0)
			{
				/* Fill tcp-specifics */
				uintSwapped = SWAPUINT(inst->TransactionId);
				memcpy(&(inst->SendBuffer[0]), &uintSwapped, 2); 								/* Transaction ID: 2 byte */
				uintSwapped = 0;
				memcpy(&(inst->SendBuffer[2]), &uintSwapped, 2); 								/* Protocol id: 2 byte */
				uintSwapped = SWAPUINT(inst->FB_MB_CreateClientRequest.RequestBufferLen + 1);
				memcpy(&inst->SendBuffer[4], &uintSwapped, 2); 									/* Length: 2 bytes */
				inst->SendBuffer[6] = inst->FB_MB_CreateClientRequest.Unit;						/* Unit: 1 byte */
				/* 7... Modbus message */
				/* Filled in by FB_MB_CreateClientRequest */
				inst->FB_TcpSend.datalen = 7 + inst->FB_MB_CreateClientRequest.RequestBufferLen;
				inst->Step = 30;

				if (!inst->Enable)
					inst->Step = 10;
			}
			else if (inst->FB_MB_CreateClientRequest.Status == 0 && inst->ConnectionTimeout > 0 && inst->ElapsedTime >= inst->ConnectionTimeout && BRSE_MBT_ClientInternal.TcpOpenIdent[inst->ClientID] != 0) /* queue empty disconnect client at timeout */
			{
				inst->Step = 70; /* close inactive client connection */
				inst->ElapsedTime = 0;
			}
			else
			{
				inst->Status = inst->FB_MB_CreateClientRequest.Status;
				if (!inst->Enable)
					inst->Step = 10;
			}
			if (inst->Step != 30)
				break;

		case 30:
			if (BRSE_MBT_ClientInternal.TcpOpenIdent[inst->ClientID] == 0) /* port not open */
				inst->Step = 31;
			else
				inst->Step = 40;

			if (inst->Step != 31)
				break;
			/* beware: fall-through on state 31 */

		case 31: /* open port */
			TcpOpen(&inst->FB_TcpOpen);
			if (inst->FB_TcpOpen.status == 0)
			{
				BRSE_MBT_ClientInternal.TcpOpenIdent[inst->ClientID] = inst->FB_TcpOpen.ident;
				inst->FB_TcpClient.ident = BRSE_MBT_ClientInternal.TcpOpenIdent[inst->ClientID];
				inst->FB_TcpClient.pServer = (UDINT)inst->IpAddr;
				inst->FB_TcpClient.portserv = inst->Port;
				inst->FB_TcpRecive.ident = BRSE_MBT_ClientInternal.TcpOpenIdent[inst->ClientID];
				inst->FB_TcpSend.ident = BRSE_MBT_ClientInternal.TcpOpenIdent[inst->ClientID];
				inst->Step = 32;
			}
			else if (inst->FB_TcpOpen.status == tcpERR_SOCKET_CREATE)  /* just wait for a socket */
			{
				;
			}
			else if (inst->FB_TcpOpen.status != BUSY) /* error, close down and return error on request */
			{
				inst->ErrorStatus = inst->FB_TcpOpen.status;
				inst->Step = 90;
				inst->Timeout = 0;
			}
			break;

		case 32: /* linger options */
			inst->LingerOptions.lOnOff = 1;
			inst->LingerOptions.lLinger = inst->SocketTimeout;
			inst->FB_TcpIoctl.ident = BRSE_MBT_ClientInternal.TcpOpenIdent[inst->ClientID];
			inst->FB_TcpIoctl.ioctl = tcpSO_LINGER_SET;
			inst->FB_TcpIoctl.pData = (UDINT)&inst->LingerOptions;
			inst->FB_TcpIoctl.datalen = sizeof(inst->LingerOptions);
			TcpIoctl(&inst->FB_TcpIoctl);
			if (inst->FB_TcpIoctl.status != BUSY)
			{
				inst->Step = 33;
			}
			break;

		case 33: /* client */
			TcpClient(&inst->FB_TcpClient);
			if(inst->FB_TcpClient.status == 0)
			{
				inst->Step = 40;
			}
			else if (inst->FB_TcpClient.status != BUSY) /* error, close down and return error on request */
			{
				inst->ErrorStatus = inst->FB_TcpClient.status;
				inst->Step = 90;
			}
			break;

		case 40: /* Send request */
			inst->FB_TcpSend.enable = 1;
			TcpSend(&inst->FB_TcpSend);
			if ( (inst->FB_TcpSend.status == BUSY) ||
					(inst->FB_TcpSend.status == tcpERR_WOULDBLOCK) ||
					(inst->FB_TcpSend.status == tcpERR_SENTLEN))
			{
				;
			}
			else if (inst->FB_TcpSend.status == 0)
			{
				inst->Step = 41;
				inst->ElapsedTime = 0;
			}
			else /* Error sending request */
			{
				inst->ErrorStatus = inst->FB_TcpSend.status;
				inst->Step = 90;
			}
			break;

		case 41: /* Receive response */
			inst->ElapsedTime += inst->CycleTimeMs;
			TcpRecv(&inst->FB_TcpRecive);
			if( (inst->FB_TcpRecive.status == BUSY				) 	||
				(inst->FB_TcpRecive.status == DISABLE			)	)
			{
				;
			}
			else if (inst->FB_TcpRecive.status == tcpERR_NO_DATA) /* send timeout */
			{
				if (inst->ElapsedTime > MBT_RECEIVE_TIMEOUT && inst->ResendCounter <= BRSE_MBT_RESEND_LIMIT)
				{
					inst->ResendCounter++;
					inst->Step = 40; /* re-send */
				}
				else if (inst->ElapsedTime > MBT_RECEIVE_TIMEOUT)
				{
					inst->Step = 90; /* failed, no response */
				}
			}
			else if(inst->FB_TcpRecive.status == 0)
			{
				if(inst->FB_TcpRecive.recvlen > 8 && inst->FB_TcpRecive.recvlen < (BRSE_MBT_MAX_BUFFER+1))
				{
					memcpy(&uintSwapped, &(inst->ReceiveBuffer[0]), sizeof(uintSwapped));
					inst->RecvTransactionId = SWAPUINT(uintSwapped);
					if (inst->RecvTransactionId == inst->TransactionId)
					{
						if (inst->ReceiveBuffer[2] != 0 || inst->ReceiveBuffer[3] != 0 || (inst->ReceiveBuffer[4] == 0 && inst->ReceiveBuffer[5] == 0) )
						{
							inst->Step = 51; /* Illegal response */
						}
						else
						{
							memcpy(&uintSwapped, &(inst->ReceiveBuffer[4]), 2);
							inst->RecvLen = SWAPUINT(uintSwapped);
							inst->Step = 50; /* Put answer */
						}
					}
				}
				else if (inst->FB_TcpRecive.recvlen == 0) /* other side performed a tcp close. return error on request */
				{
					inst->Step = 90;
				}
				else
				{
					inst->Step = 51;
				}
			}
			else
			{
				inst->ErrorStatus = inst->FB_TcpRecive.status;
				inst->Step = 90;
			}
			break;

		case 50: /* put response */
			inst->FB_MB_PutClientResponse.AdrByteBuffer = (UDINT)&(inst->ReceiveBuffer[7]);
			inst->FB_MB_PutClientResponse.ByteBufferLen = inst->RecvLen -1 ;
			inst->FB_MB_PutClientResponse.ClientID = inst->ClientID;
			inst->FB_MB_PutClientResponse.ServerFormat = inst->ServerFormat;
			MB_PutClientResponse(&inst->FB_MB_PutClientResponse);
			if (inst->FB_MB_PutClientResponse.Status != BUSY) /* ok, done. does not matter if error or not. */
			{
				memset(&(inst->SendBuffer[0]), 0, sizeof(inst->SendBuffer));
				inst->Step = 10;
				inst->TransactionId++;
			}
			break;

		case 51: /* put error response */
			memset(&(inst->SendBuffer[0]), 0, sizeof(inst->SendBuffer));
			inst->Status = MB_AckClientRequest(inst->ClientID, MB_ERR_PROTOCOL);
			if (inst->Status != BUSY)
			{
				inst->Step = 10;
				inst->TransactionId++;
			}
			break;

		case 70: /* disconnect inactive client connection */
			inst->FB_TcpClose.ident	= BRSE_MBT_ClientInternal.TcpOpenIdent[inst->ClientID];
			inst->FB_TcpClose.how = 0;
			TcpClose(&inst->FB_TcpClose);
			if(inst->FB_TcpClose.status != BUSY)
			{
				BRSE_MBT_ClientInternal.TcpOpenIdent[inst->ClientID] = 0;
				inst->Step = 10;
			}
			break;

		case 90: /* Error */
			if (BRSE_MBT_ClientInternal.TcpOpenIdent[inst->ClientID] == 0)
			{
				inst->Step = 91;
			}
			else
			{
				inst->FB_TcpClose.ident	= BRSE_MBT_ClientInternal.TcpOpenIdent[inst->ClientID];
				inst->FB_TcpClose.how = 0;
				TcpClose(&inst->FB_TcpClose);
				if(inst->FB_TcpClose.status != BUSY)
				{
					BRSE_MBT_ClientInternal.TcpOpenIdent[inst->ClientID] = 0;
					inst->Step = 91;
				}
			}
			break;

		case 91:
			memset(&(inst->SendBuffer[0]), 0, sizeof(inst->SendBuffer));
			inst->Status = MB_AckClientRequest(inst->ClientID, MB_ERR_CONNECTION);
			if (inst->Status != BUSY)
			{
				inst->Step = 10;
				inst->TransactionId++;
			}
			break;
	}
}

/*!
	\interface MBT_ExitClient
	\brief Client: Closes open tcp ports. Use this in the exit routine of the program.

	\param[in] 	ClientID	Identity created in AllocClient.
	\param[out] Status	Return status.

*/
void MBT_ExitClient(struct MBT_ExitClient* inst)
{
	if (BRSE_MBT_ClientInternal.TcpOpenIdent[inst->ClientID] != 0)
	{
		inst->FB_TcpClose.enable = 1;
		inst->FB_TcpClose.ident	= BRSE_MBT_ClientInternal.TcpOpenIdent[inst->ClientID];
		inst->FB_TcpClose.how = tcpSHUT_RD | tcpSHUT_WR;
		TcpClose(&inst->FB_TcpClose);
		if(inst->FB_TcpClose.status != BUSY)
		{
			BRSE_MBT_ClientInternal.TcpOpenIdent[inst->ClientID] = 0;
		}
	}
}
```

#### Version_History.c
```c
/*! \file Version_History.c */

/*!
\page History

\section History

\par V0.00
	\arg First draft version

\par V1.00
	\arg First functional version. Added inline comments.

\par V1.01
	\arg Removed the input Unit in the MBT_client. Make it possible to communicate to many units in the same server in a simple way.
	\arg Added documentation for the client.

\par V1.02
	\arg Updated documentation.

\par V1.03
	\arg Added functionality for handling 4 byte variables.

\par V1.10
	\arg release version including 4 byte holding registers.
	\arg bugfix for client which previously used up all idents if server was unavailable.

\par V1.11
	\arg BRSE_MB_Server function has been rewritten to improve performance. Requests from each client are now responded to in the same cycle.
	\arg That brings the execution time to depend very much on the server load, i.e. frequency of client requests

\par V1.12
	\arg Bugfixes:
	\arg If timeout occurs during TcpRecv, the FUB is only aborted if tcpERR_NO_DATA is the status.
	\arg The timeout in TcpClient has been removed, since it was unnecessary and aborted TcpClient during execution.
	\arg On the server side, if error code tcpERR_SENTLEN is received, it retries sending instead of disconnecting the client.

\par V1.13
	\arg New feature: ConnectionMode for client. Default behaviour: When the queue is empty, the connection is closed. Optional behaviour: the connection statys open.
	\arg Bugfixed: Stability improvements in both server and clients. Reconneciton-patterns and error behaviours have been revised.
\par V1.14
	\arg MAX_CLIENTS has been set up to 10, as this is above the socket limit for SGC CPUs.
	\arg BRSE_MBT_Server / MBT_Client : new input \b SocketTimeout which specifies the time for the system to close down the socket (see also AsTCP linger set) in seconds.
	\arg MBT_Client : New input \b ConnectionTimeout, has replaced the input \b ConnectionMode, and now specifies the time until an empty queue closes the connection to the server.
	\arg MBT_Client : Changed behaviour when a server does not respond to a request. Before, the client would retry to send the request, but now the client just passes on an error message to the corresponding BRSE_MB block.
	\arg Added dependency to the brsystem library, which reads out the cycle time of the task. In this way, the MBT_Client is no longer dependent on the \b CycleTime input. It has therefore been removed.
\par V1.15
	\arg MBT_Client, BRSE_MBT_Server : Changed behaviour of the SocketTimeout input when it is zero. Value Zero now disables lingering, the connection closes immediately.
\par V1.20
	\arg BRSE_MBT_Server : Bugfix for closing connections. There was a problem when closing many clients simultaneously which left sockets open.
	The cause of the error was that only one instance of the tcpclose function was used.
	Now there are BRSE_MBT_MAX_CLIENTS instances of TcpClose, which solves this error.
*/
```

### Program Logical/ExtPack/_Comms/SNTPClient/SNTPClient_v1/NwSNTPClient (IEC) - SNTP client configuration

#### NwSNTPClient.st - Implementation code
```iecst
(********************************************************************
 * COPYRIGHT -- Bernecker + Rainer
 ********************************************************************
 * Program: NwSNTPClient
 * File: NwSNTPClient.st
 * Author: Bernecker + Rainer
 * Created: April 21, 2009
 ********************************************************************
 * Implementation of program NwSNTPClient
 ********************************************************************)

PROGRAM _INIT

	Time ACCESS ADR(gTime);

	(* Init values *)
	strcpy(ADR(Network.Data.SNTPServerAddress),ADR('192.168.127.50'));  (* IP address of the SNTP server *)

	Network.Data.SNTPInterval := 1;
	Network.Data.RTCInterval := 2;

	Network.Data.TimeZoneYear := 2022;

END_PROGRAM

PROGRAM _CYCLIC

	//Define the proper TimeZoneId with the UTC TimeZone and the
	TimeStateMachine;

	CASE Network.Data.Step OF

		0:	IF Network.Command.bCfgGetSntpcData = 1 THEN
  				Network.Data.Step := 10;
			ELSIF Network.Command.bCfgSetSntpClient = 1 THEN
				Network.Data.Step := 20;
			ELSIF Network.Command.bGetTimeData = 1 THEN
				Network.Data.Step := 30;
			ELSIF Network.Command.bCfgSetTimeOffset = 1 THEN
				Network.Data.Step := 70;
			ELSIF Network.Command.bCfgSetDst = 1 THEN
				Network.Data.Step := 80;
			ELSIF Network.Command.bCfgSetTimeZone = 1 THEN
				Network.Data.Step := 90;
			END_IF

		10:  (* Get the parameters relevant for the SNTP client *)
			Network.Functionblocks.CfgGetSntpcData_0.enable := 1;  (* Enable the function block *)
			Network.Functionblocks.CfgGetSntpcData_0.pServerAddr := ADR(Network.Data.SNTPServerAddress);  (* IP address of the SNTP server *)
			Network.Functionblocks.CfgGetSntpcData_0.Len := SIZEOF(Network.Data.SNTPServerAddress);  (* Length of the SNTP server address string *)

			Network.Functionblocks.CfgGetSntpcData_0;  (* Function Call *)

			IF Network.Functionblocks.CfgGetSntpcData_0.status = 0 THEN  (* CfgGetSntpcData successfull *)
				Network.Data.SNTPStatus := Network.Functionblocks.CfgGetSntpcData_0.run;
				Network.Data.SNTPInterval := Network.Functionblocks.CfgGetSntpcData_0.sntpcInterval;
				Network.Data.RTCInterval := Network.Functionblocks.CfgGetSntpcData_0.rtcInterval;
				Network.Command.bCfgGetSntpcData := 0;
				Network.Data.Step := 0;
			ELSIF Network.Functionblocks.CfgGetSntpcData_0.status = ERR_FUB_BUSY THEN  (* CfgGetSntpcData not finished -> redo *)
				(* Busy *)
			ELSE  (* Goto Error Step *)
				Network.Data.Step := 255;
			END_IF

		20:  (* Configure, start, or stop the SNTP client *)
			Network.Functionblocks.CfgSetSntpClient_0.enable := 1;  (* Enable the function block *)
			Network.Functionblocks.CfgSetSntpClient_0.run := 1;  (* Start the SNTP client *)
			Network.Functionblocks.CfgSetSntpClient_0.pServerAddr := ADR(Network.Data.SNTPServerAddress);  (* IP address of the SNTP server *)
			Network.Functionblocks.CfgSetSntpClient_0.sntpcInterval := Network.Data.SNTPInterval;  (* Interval for the SNTP client to synchronize the time with the server *)
			Network.Functionblocks.CfgSetSntpClient_0.rtcInterval := Network.Data.RTCInterval;  (* Interval for the RTC and software time synchronization *)
			Network.Functionblocks.CfgSetSntpClient_0.option := cfgOPTION_VOLATILE;  (*  Temporarily set the parameter *)

			Network.Functionblocks.CfgSetSntpClient_0;  (* Function Call *)

			IF Network.Functionblocks.CfgSetSntpClient_0.status = 0 THEN  (* CfgSetSntpClient successfull *)

				Network.Data.SyncStatus := Network.Functionblocks.CfgSetSntpClient_0.syncStatus;

				IF Network.Functionblocks.CfgSetSntpClient_0.syncStatus = 2 THEN  (* Client active and time received at least once from server *)
					Network.Command.bCfgSetSntpClient := 0;
					Network.Data.Step := 0;
				ELSIF Network.Functionblocks.CfgSetSntpClient_0.syncStatus = 1 THEN  (* Client already active, but time not received from server *)
					Network.Command.bCfgSetSntpClient := 0;
					Network.Data.Step := 0;
				ELSE  (* Client not active *)
					Network.Data.Step := 255;
				END_IF

			ELSIF Network.Functionblocks.CfgSetSntpClient_0.status = ERR_FUB_BUSY THEN  (* CfgSetSntpClient not finished -> redo *)
				(* Busy *)
			ELSE  (* Goto Error Step *)
				Network.Data.Step := 255;
			END_IF

		30:  (* Get the configured time offset *)
			Network.Functionblocks.CfgGetTimeOffset_0.enable := 1;  (* Enable the function block *)

			Network.Functionblocks.CfgGetTimeOffset_0;  (* Function Call *)

			IF Network.Functionblocks.CfgGetTimeOffset_0.status = 0 THEN  (* CfgGetTimeOffset successfull *)
				Network.Data.TimeOffset := Network.Functionblocks.CfgGetTimeOffset_0.timeoffset;
				Network.Data.Step := 40;
			ELSIF Network.Functionblocks.CfgGetTimeOffset_0.status = ERR_FUB_BUSY THEN  (* CfgGetTimeOffset not finished -> redo *)
				(* Busy *)
			ELSE  (* Goto Error Step *)
				Network.Data.Step := 255;
			END_IF

		40:  (* Get the ID of the currently active timezone *)
			Network.Functionblocks.CfgGetTimeZone_0.enable := 1;  (* Enable the function block *)

			Network.Functionblocks.CfgGetTimeZone_0;  (* Function Call *)

			IF Network.Functionblocks.CfgGetTimeZone_0.status = 0 THEN  (* CfgGetTimeZone successfull *)
				Network.Data.TimeZoneID := Network.Functionblocks.CfgGetTimeZone_0.timezoneID;
				Network.Data.Step := 50;
			ELSIF Network.Functionblocks.CfgGetTimeZone_0.status = ERR_FUB_BUSY THEN  (* CfgGetTimeZone not finished -> redo *)
				(* Busy *)
			ELSE  (* Goto Error Step *)
				Network.Data.Step := 255;
			END_IF

		50:  (* Get the times when the time switches for a particular timezone in a specified year *)
			Network.Functionblocks.CfgGetTimeZoneEntry_0.enable := 1;  (* Enable the function block *)
			Network.Functionblocks.CfgGetTimeZoneEntry_0.timezoneID := Network.Data.TimeZoneID;
			Network.Functionblocks.CfgGetTimeZoneEntry_0.year := Network.Data.TimeZoneYear;

			Network.Functionblocks.CfgGetTimeZoneEntry_0;  (* Function Call *)

			IF Network.Functionblocks.CfgGetTimeZoneEntry_0.status = 0 THEN  (* CfgGetTimeZoneEntry successfull *)
				Network.Data.DateSummerTime := Network.Functionblocks.CfgGetTimeZoneEntry_0.dateDst;
				Network.Data.DateNormalTime := Network.Functionblocks.CfgGetTimeZoneEntry_0.dateNormal;
				Network.Data.Step := 60;
			ELSIF Network.Functionblocks.CfgGetTimeZoneEntry_0.status = ERR_FUB_BUSY THEN  (* CfgGetTimeZoneEntry not finished -> redo *)
				(* Busy *)
			ELSE  (* Goto Error Step *)
				Network.Data.Step := 255;
				Network.Functionblocks.CfgGetTimeZoneEntry_0.enable := 0;  (* Disanble the function block *)
				Network.Functionblocks.CfgGetTimeZoneEntry_0;  (* Function Call *)
			END_IF

		60:  (* Get the time offset between a timezone and GMT during normal time (gmt) and during summer time (gmtDst) *)
			Network.Functionblocks.CfgGetTimeZoneInfo_0.enable := 1;  (* Enable the function block *)
			Network.Functionblocks.CfgGetTimeZoneInfo_0.timezoneID := Network.Data.TimeZoneID;

			Network.Functionblocks.CfgGetTimeZoneInfo_0;  (* Function Call *)

			IF Network.Functionblocks.CfgGetTimeZoneInfo_0.status = 0 THEN  (* CfgGetTimeZoneInfo successfull *)
				Network.Data.DeviationGMT := Network.Functionblocks.CfgGetTimeZoneInfo_0.gmt;
				Network.Data.DeviationGMTDst := Network.Functionblocks.CfgGetTimeZoneInfo_0.gmtDst;
				Network.Command.bGetTimeData := 0;
				Network.Data.Step := 0;
			ELSIF Network.Functionblocks.CfgGetTimeZoneInfo_0.status = ERR_FUB_BUSY THEN  (* CfgGetTimeZoneInfo not finished -> redo *)
				(* Busy *)
			ELSE  (* Goto Error Step *)
				Network.Data.Step := 255;
				Network.Functionblocks.CfgGetTimeZoneInfo_0.enable := 0;  (* Disanble the function block *)
				Network.Functionblocks.CfgGetTimeZoneInfo_0;  (* Function Call *)
			END_IF

		70:  (* Set a time offset *)
			Network.Functionblocks.CfgSetTimeOffset_0.enable := 1;  (* Enable the function block *)
			Network.Functionblocks.CfgSetTimeOffset_0.timeoffset := Network.Data.TimeOffset;  (* Time offset to be configured [minutes] *)
			Network.Functionblocks.CfgSetTimeOffset_0.option := cfgOPTION_VOLATILE;  (*  Temporarily set the parameter *)

			Network.Functionblocks.CfgSetTimeOffset_0;  (* Function Call *)

			IF Network.Functionblocks.CfgSetTimeOffset_0.status = 0 THEN  (* CfgSetTimeOffset successfull *)
				Network.Command.bCfgSetTimeOffset := 0;
				Network.Data.Step := 0;
			ELSIF Network.Functionblocks.CfgSetTimeOffset_0.status = ERR_FUB_BUSY THEN  (* CfgSetTimeOffset not finished -> redo *)
				(* Busy *)
			ELSE  (* Goto Error Step *)
				Network.Data.Step := 255;
				Network.Functionblocks.CfgSetTimeOffset_0.enable := 0;  (* Disaable the function block *)
				Network.Functionblocks.CfgSetTimeOffset_0;  (* Function Call *)
			END_IF

		80:  (* Enable or disable automatic daylight savings time *)
			Network.Functionblocks.CfgSetDst_0.enable := 1;  (* Enable the function block *)
			Network.Functionblocks.CfgSetDst_0.dst := 1;  (* enables automatic daylight savings time *)
			Network.Functionblocks.CfgSetDst_0.option := cfgOPTION_VOLATILE;  (*  Temporarily set the parameter *)

			Network.Functionblocks.CfgSetDst_0;  (* Function Call *)

			IF Network.Functionblocks.CfgSetDst_0.status = 0 THEN  (* CfgSetDst successfull *)
				Network.Command.bCfgSetDst := 0;
				Network.Data.Step := 0;
			ELSIF Network.Functionblocks.CfgSetDst_0.status = ERR_FUB_BUSY THEN  (* CfgSetDst not finished -> redo *)
				(* Busy *)
			ELSE  (* Goto Error Step *)
				Network.Data.Step := 255;
			END_IF

		90:  (* Set the time zone *)
			Network.Functionblocks.CfgSetTimeZone_0.enable := 1;  (* Enable the function block *)
			Network.Functionblocks.CfgSetTimeZone_0.timezoneID := Network.Data.TimeZoneID;  (* ID of the timezone you would like to set *)
			Network.Functionblocks.CfgSetTimeZone_0.option := cfgOPTION_VOLATILE;  (*  Temporarily set the parameter *)

			Network.Functionblocks.CfgSetTimeZone_0;  (* Function Call *)

			IF Network.Functionblocks.CfgSetTimeZone_0.status = 0 THEN  (* CfgSetTimeZone successfull *)
				Network.Command.bCfgSetTimeZone := 0;
				Network.Data.Step := 0;
			ELSIF Network.Functionblocks.CfgSetTimeZone_0.status = ERR_FUB_BUSY THEN  (* CfgSetTimeZone not finished -> redo *)
				(* Busy *)
			ELSE  (* Goto Error Step *)
				Network.Data.Step := 255;
			END_IF

	END_CASE

END_PROGRAM
```

#### TimeZoneId.st
```iecst
ACTION TimeZoneId:

	CASE Time.Params.UTCTimeZone OF
		-1200: Network.Data.TimeZoneID := 5;
		-1100: Network.Data.TimeZoneID := 10;
		-1000: Network.Data.TimeZoneID := 15;
		-0900: Network.Data.TimeZoneID := 20;
		-0800: Network.Data.TimeZoneID := 25;
		-0700: IF Time.Params.DayLightSavingsTime THEN Network.Data.TimeZoneID := 35; ELSE Network.Data.TimeZoneID := 30; END_IF
		-0600: IF Time.Params.DayLightSavingsTime THEN Network.Data.TimeZoneID := 45; ELSE Network.Data.TimeZoneID := 55; END_IF
		-0500: IF Time.Params.DayLightSavingsTime THEN Network.Data.TimeZoneID := 65; ELSE Network.Data.TimeZoneID := 60; END_IF
		-0400: IF Time.Params.DayLightSavingsTime THEN Network.Data.TimeZoneID := 85; ELSE Network.Data.TimeZoneID := 80; END_IF
		-0330: Network.Data.TimeZoneID := 95;
		-0300: IF Time.Params.DayLightSavingsTime THEN Network.Data.TimeZoneID := 105; ELSE Network.Data.TimeZoneID := 110; END_IF
		-0200: Network.Data.TimeZoneID := 115;
		-0100: IF Time.Params.DayLightSavingsTime THEN Network.Data.TimeZoneID := 120; ELSE Network.Data.TimeZoneID := 125; END_IF
		0000:  IF Time.Params.DayLightSavingsTime THEN Network.Data.TimeZoneID := 130; ELSE Network.Data.TimeZoneID := 135; END_IF
		+0100: IF Time.Params.DayLightSavingsTime THEN Network.Data.TimeZoneID := 140; ELSE Network.Data.TimeZoneID := 155; END_IF
		+0200: IF Time.Params.DayLightSavingsTime THEN Network.Data.TimeZoneID := 165; ELSE Network.Data.TimeZoneID := 180; END_IF
		+0300: Network.Data.TimeZoneID := 200;
		+0330: Network.Data.TimeZoneID := 215;
		+0400: IF Time.Params.DayLightSavingsTime THEN Network.Data.TimeZoneID := 230; ELSE Network.Data.TimeZoneID := 220; END_IF
		+0430: Network.Data.TimeZoneID := 235;
		+0500: Network.Data.TimeZoneID := 240;
		+0530: Network.Data.TimeZoneID := 250;
		+0545: Network.Data.TimeZoneID := 255;
		+0600: Network.Data.TimeZoneID := 260;
		+0630: Network.Data.TimeZoneID := 280;
		+0700: Network.Data.TimeZoneID := 285;
		+0800: Network.Data.TimeZoneID := 295;
		+0900: Network.Data.TimeZoneID := 320;
		+0930: Network.Data.TimeZoneID := 335;
		+1000: IF Time.Params.DayLightSavingsTime THEN Network.Data.TimeZoneID := 350; ELSE Network.Data.TimeZoneID := 340; END_IF
		+1100: Network.Data.TimeZoneID := 365;
		+1200: IF Time.Params.DayLightSavingsTime THEN Network.Data.TimeZoneID := 370; ELSE Network.Data.TimeZoneID := 375; END_IF
		+1300: Network.Data.TimeZoneID := 380;

	END_CASE;

END_ACTION
```

#### NwSNTPClient.typ - Local data types
```iecst
(********************************************************************
 * COPYRIGHT -- Bernecker + Rainer
 ********************************************************************
 * Program: NwSNTPClient
 * File: NwSNTPClient.typ
 * Author: Bernecker + Rainer
 * Created: April 21, 2009
 ********************************************************************
 * Local data types of program NwSNTPClient
 ********************************************************************)

TYPE
	SNTP_Network_typ : 	STRUCT
		Command : SNTP_Network_Command_typ; (*Structure Command (contains all command elements)*)
		Data : SNTP_Network_Data_typ; (*Structure Data (contains all data informations)*)
		Functionblocks : SNTP_Network_Functionblocks_typ; (*Structure Functionblocks (contains all FuBs)*)
	END_STRUCT;
	SNTP_Network_Command_typ : 	STRUCT
		bCfgGetSntpcData : BOOL; (*Command: Get SNTP client data*)
		bGetTimeData : BOOL; (*Command: Get several time data*)
		bCfgSetSntpClient : BOOL; (*Command: Start SNTP client*)
		bCfgSetTimeOffset : BOOL; (*Command: Set the configured time offset*)
		bCfgSetDst : BOOL; (*Command: Enable the automatic daylight savings time*)
		bCfgSetTimeZone : BOOL; (*Command: Set the configured time zone*)
	END_STRUCT;
	SNTP_Network_Data_typ : 	STRUCT
		SNTPServerAddress : STRING[16]; (*Data variable for CfgGetSntpcData() and CfgSetSntpClient()*)
		SNTPStatus : UDINT; (*Data variable for CfgGetSntpcData()*)
		SNTPInterval : UINT; (*Data variable for CfgGetSntpcData() and CfgSetSntpClient()*)
		RTCInterval : UINT; (*Data variable for CfgGetSntpcData() and CfgSetSntpClient()*)
		SyncStatus : USINT; (*Data variable for CfgSetSntpClient()*)
		TimeOffset : UINT; (*Data variable for CfgGetTimeOffset() and CfgSetTimeOffset()*)
		TimeZoneID : UINT; (*Data variable for CfgGetTimeZone(), CfgGetTimeZoneEntry(), CfgGetTimeZoneInfo() and CfgSetTimeZone()*)
		TimeZoneYear : UINT; (*Data variable for CfgGetTimeZoneEntry()*)
		DateSummerTime : DATE_AND_TIME; (*Data variable for CfgGetTimeZoneEntry()*)
		DateNormalTime : DATE_AND_TIME; (*Data variable for CfgGetTimeZoneEntry()*)
		DeviationGMT : UINT; (*Data variable for CfgGetTimeZoneInfo()*)
		DeviationGMTDst : UINT; (*Data variable for CfgGetTimeZoneInfo()*)
		Step : USINT; (*Step variable*)
	END_STRUCT;
	SNTP_Network_Functionblocks_typ : 	STRUCT
		CfgGetSntpcData_0 : CfgGetSntpcData; (*Functionblock CfgGetSntpcData()*)
		CfgSetSntpClient_0 : CfgSetSntpClient; (*Functionblock CfgSetSntpClient()*)
		CfgGetTimeOffset_0 : CfgGetTimeOffset; (*Functionblock CfgGetTimeOffset()*)
		CfgGetTimeZone_0 : CfgGetTimeZone; (*Functionblock CfgGetTimeZone()*)
		CfgGetTimeZoneEntry_0 : CfgGetTimeZoneEntry; (*Functionblock CfgGetTimeZoneEntry()*)
		CfgGetTimeZoneInfo_0 : CfgGetTimeZoneInfo; (*Functionblock CfgGetTimeZoneInfo()*)
		CfgSetTimeOffset_0 : CfgSetTimeOffset; (*Functionblock CfgSetTimeOffset()*)
		CfgSetDst_0 : CfgSetDst; (*Functionblock CfgSetDst()*)
		CfgSetTimeZone_0 : CfgSetTimeZone; (*Functionblock CfgSetTimeZone()*)
	END_STRUCT;
END_TYPE
```

#### NwSNTPClient.var - Local variables
```iecst
(********************************************************************
 * COPYRIGHT -- Bernecker + Rainer
 ********************************************************************
 * Program: NwSNTPClient
 * File: NwSNTPClient.var
 * Author: Bernecker + Rainer
 * Created: April 21, 2009
 ********************************************************************
 * Local variables of program NwSNTPClient
 ********************************************************************)
VAR
	Network : {REDUND_UNREPLICABLE} SNTP_Network_typ; (*Global structure*)
	Time : REFERENCE TO TimeMachine;
	TimeZoneId_copy : UINT;
	xNeedToResedTimeZoneId : BOOL;
END_VAR
```

- SNTP Configuration. PressPC & PLC.docx (binary file, 1797182 bytes)
### Feeder.typ
```iecst
TYPE
	FeederCtrlStatus_enum :
		(
		FEEDERCTRL_STOPPED,
		FEEDERCTRL_STOPPING,
		FEEDERCTRL_PREPARING,
		FEEDERCTRL_PREPARED,
		FEEDERCTRL_PAUSING,
		FEEDERCTRL_PAUSED,
		FEEDERCTRL_STARTING,
		FEEDERCTRL_FEEDING,
		FEEDERCTRL_CONTROLSTOPPING
		);
	FeederStatus_enum :
		(
		FEEDER_TURNED_OFF,
		FEEDER_INIT,
		FEEDER_PREPARING,
		FEEDER_READY,
		FEEDER_FEEDING,
		FEEDER_FAULTED
		);
	FeederType_enum :
		(
		FEEDERTY_UNDEFINED,
		FEEDERTY_BOTTOM_14, (*Bottom feeder. Serra manufacturer. 1400mm width*)
		FEEDERTY_BOTTOM_18, (*Bottom feeder. Serra manufacturer. 1800mm width*)
		FEEDERTY_TOP (*Top feeder. BDT manufacturer. 1800mm width*)
		);
	FeederInputs_typ : 	STRUCT
		xOnline : BOOL;
		xError : BOOL;
		xFeeding : BOOL;
		xMultiPick : BOOL; (*BDT Feeder specifi signal*)
		xTrayEmpty : BOOL;
		xFeederPresent : BOOL;
		xMediaThickness : BOOL;
		xReadyToFeed : BOOL;
		xMediaLowL1 : BOOL;
		xMediaLowL2 : BOOL;
		xJamDetection : BOOL; (*SerraFeeder specific signal.*)
		xTrayEmptyL1 : BOOL;
		xTrayEmptyL2 : BOOL;
		xModelInput : ARRAY[0..2]OF BOOL;
		xNoPowered : BOOL;
		Comms : FeederCommsInputs_typ;
	END_STRUCT;
	FeederOutputs_typ : 	STRUCT
		Physical : FeederPhysicalOutputs_typ;
		Comms : FeederCommsOutputs_typ;
	END_STRUCT;
	FeederAlarms_typ : 	STRUCT
		xError : BOOL;
		xNotOnline : BOOL;
		xNotRemote : BOOL;
		xNoFeederPresent : BOOL;
		xAnyAlarm : BOOL;
		xMediaLowL1 : BOOL;
		xMediaLowL2 : BOOL;
		xTrayEmptyL1 : BOOL;
		xTrayEmptyL2 : BOOL;
		xNoPowered : BOOL;
		xCriticalAlarm : BOOL;
		xWarningAlarm : BOOL;
		xCommsError : BOOL;
		xStopRequest : BOOL; (*Stop request from Dryer when physical stop button is pressed*)
	END_STRUCT;
	FeederParametersSw_typ : 	STRUCT
		xEnabled : BOOL;
		xBatchFeeding : BOOL; (*1:Batch feeding mode; 0: continuous feeding.*)
		iCentralOffset : INT; (*Offset value received from SW for feeders with Parameters.Hw.xOffsetAvailable = TRUE;*)
	END_STRUCT;
	FeederParametersHw_typ : 	STRUCT
		iMaxMediaWidth : UINT; (*Maximum media width allowed in mm*)
		iMinMediaWidth : UINT; (*Minimum media width allowed in mm*)
		iMinMediaLength : UINT; (*Minimum media length allowed in mm*)
		iMaxMediaLength : UINT; (*Maximum media length allowed in mm*)
		xOffsetAvailable : BOOL; (*Offset line alignment parameter available*)
		iMaxOffset : UINT; (*Upper limit for line alignment offset value [mm]*)
		iMinOffset : INT; (*Lower limit for line alignment offset value [mm]*)
		iMinMediaThickness : UINT; (*Minimum media height allowed in tenth of mm*)
		iMaxMediaThickness : UINT; (*Maximum media height allowed in tenth of mm*)
		rMaxSpeed : REAL := 100.0; (*Maximum speed allowed in m/min*)
		xDoubleLineAllowed : BOOL; (*Active when printer allows double line printing*)
	END_STRUCT;
	FeederParameters_typ : 	STRUCT
		xInstalled : BOOL;
		xSimulationMode : BOOL; (*Defined by the configuration in Automation Studio*)
		xCommsOK : BOOL;
		xAlrPresent : BOOL;
		LineState : LineStatus_enum;
		iRegisterType : UINT := 1; (*0:lateral; 1:central*)
		iLineConfig : UINT;
		xLineInAuto : BOOL;
		Media : FeederMediaParameters;
		rBeltSpeedSetPoint : REAL;
		xDoubleLine : BOOL;
		iCentralOffset : INT; (*(-500, 500) Limis*)
		iCounterSetPointL1 : INT;
		iCounterSetPointL2 : INT;
		LineStatusSummary : LineControlStatusSummarized;
		Hw : FeederParametersHw_typ;
		xActiveSlaveDiagnosis : BOOL;
	END_STRUCT;
	FeederCommands_typ : 	STRUCT
		xBelEmpty : BOOL; (*Edge commands. Reseted when managed*)
		xStart : BOOL; (*Edge commands. Reseted when managed*)
		xPrepare : BOOL; (*Edge commands. Reseted when managed*)
		xPause : BOOL; (*Edge commands. Reseted when managed*)
		xControlStop : BOOL; (*Edge commands. Reseted when managed*)
		xStop : BOOL; (*Edge commands. Reseted when managed*)
		xStartTransport : BOOL; (*Edge commands. Reseted when managed*)
		xThereIsFeeder : BOOL;
		xResetAlarms : BOOL;
		xNewBoardParameters : BOOL; (*Set 1 when there is sent a new configuration.*)
		xNewOrder : BOOL; (*New batch. Set when there is sent a new job. This signal reset the current counter*)
		xSheetFeeding : BOOL;
		xStopFeeding : BOOL; (*This signal just stop the feeding, not stop the machine*)
	END_STRUCT;
	FeederDeviceStatus_typ : 	STRUCT
		xTurnedOff : BOOL;
		xInit : BOOL;
		xPreparing : BOOL;
		xReadyToFeed : BOOL;
		xFeeding : BOOL;
		xFaulted : BOOL;
	END_STRUCT;
	FeederStatus_typ : 	STRUCT
		iModel : USINT := 1; (*Model of the Device*)
		Version : EFI_version_typ;
		CtrlStatus : FeederCtrlStatus_enum;
		DeviceStatus : FeederStatus_enum;
		Device : FeederDeviceStatus_typ;
		FeederType : FeederType_enum;
		Comms : FeederCommsStatus_typ;
	END_STRUCT;
	Feeder_typ : 	STRUCT
		Inputs : FeederInputs_typ;
		Outputs : FeederOutputs_typ;
		Alarms : FeederAlarms_typ;
		ParSw : FeederParametersSw_typ;
		Parameters : FeederParameters_typ;
		Commands : FeederCommands_typ;
		Status : FeederStatus_typ;
		Orders : FeederOrders_typ;
	END_STRUCT;
	FeederPhysicalOutputs_typ : 	STRUCT
		xPrepareToFeed : BOOL;
		xFastStop : BOOL;
		xStartFeeding : BOOL;
	END_STRUCT;
	FeederCommsOutputs_typ : 	STRUCT
		iControl : INT; (*Status word*)
	END_STRUCT;
	FeederCommsInputs_typ : 	STRUCT
		iNumBoardsRemainingL1 : INT; (*Recirculation of the primer enabled in the device*)
		iNumBoardsRemainingL2 : INT; (*Recirculation of the primer enabled in the device*)
		iNumFedBoards : INT;
		xOnline : BOOL; (*Recirculation of the primer enabled in the device*)
		xEnableFeeding : BOOL; (*Recirculation of the primer enabled in the device*)
		xMinimumStackLevelL1 : BOOL; (*Recirculation of the primer enabled in the device*)
		xMinimumStackLevelL2 : BOOL; (*Recirculation of the primer enabled in the device*)
		xOrderEnd : BOOL; (*Recirculation of the primer enabled in the device*)
		xPositionReady : BOOL; (*Recirculation of the primer enabled in the device*)
		xAlarmPresent : BOOL; (*Recirculation of the primer enabled in the device*)
		xRemote : BOOL; (*Recirculation of the primer enabled in the device*)
		iVersion1 : INT; (*Machine platform (Nozomi = 1)*)
		iVersion2 : INT; (*Machine project (C18000 = 0 / C14000 = 1)*)
		iVersion3 : INT; (*Hardware version*)
		iVersion4 : INT; (*Sotfware version*)
		iStatus : INT; (*Status word*)
		iAlarmWord1 : INT; (*Status word*)
		iAlarmWord2 : INT; (*Status word*)
		iAlarmWord3 : INT; (*Status word*)
		iAlarmWord4 : INT; (*Status word*)
		iAlarmWord5 : INT; (*Status word*)
		iAlarmWord6 : INT; (*Status word*)
		iAlarmWord7 : INT; (*Status word*)
		iAlarmWord8 : INT; (*Status word*)
		iAlarmWord9 : INT; (*Status word*)
		iAlarmWord10 : INT; (*Status word*)
		iAlarmWord11 : INT; (*Status word*)
		iAlarmWord12 : INT; (*Status word*)
		iAlarmWord13 : INT; (*Status word*)
		iAlarmWord14 : INT; (*Status word*)
		iAlarmWord15 : INT; (*Status word*)
	END_STRUCT;
	FeederMediaParameters : 	STRUCT
		rThickness : REAL; (*Tile thickness to print from gui in mm*)
		rWidth : REAL; (*Board's width in mm*)
		rGap : REAL; (*Gap between boards in mm*)
		rLength : REAL; (*Board's length in mm*)
		rOffsetRegisterL1 : REAL; (*Board's width in mm*)
		rOffsetRegisterL2 : REAL; (*Board's width in mm*)
	END_STRUCT;
	FeederCommsStatus_typ : 	STRUCT
		xModuleOk : BOOL;
		ModSlaveState : UINT;
		LastError : UINT;
		LastErrorBlockNum : UINT;
		xStopButtonPressed : BOOL;
		ActOverloadError : BOOL;
		ActModbusError : BOOL;
		ActSlvConError : BOOL;
		ActRefreshError : BOOL;
		ActInternalError : BOOL;
		ActConfError : BOOL;
		HistOverloadError : BOOL;
		HistModbusError : BOOL;
		HistSlvConError : BOOL;
		HistRefreshError : BOOL;
		HistInternalError : BOOL;
		HistConfError : BOOL;
		ModbusErrorCnt : UINT;
		ModbusConErrorCnt : UINT;
		ModbusPktRefreshTimeoutCnt : UINT;
		ModbusPktPendPerSec : UINT;
		ModbusMeanResponseTime : UINT;
	END_STRUCT;
	FeederOrders_typ : 	STRUCT
		xDisableReadBlock : BOOL;
		xDisableWriteBlock : BOOL;
	END_STRUCT;
END_TYPE
```

### Program Logical/ExtPack/_Ancillaries/FeederCtrl/FeederCtrl_v1/FeederCtrl

#### Alarms.st
```iecst
ACTION Alarms:

	Feeder.Alarms.xNoFeederPresent:= NOT Feeder.Inputs.xFeederPresent;

	//IF NO Feeder, define that alarm and exit
	IF Feeder.Alarms.xNoFeederPresent THEN
		ResetAlarms;
		Feeder.Alarms.xNoFeederPresent:=TRUE;
	END_IF

	//Feeder No Powered Warning
	IF Feeder.Inputs.xNoPowered THEN Feeder.Alarms.xNoPowered := TRUE; END_IF

	Feeder.Alarms.xTrayEmptyL1 := Feeder.Inputs.xTrayEmptyL1;
	Feeder.Alarms.xMediaLowL1 := Feeder.Inputs.xMediaLowL1;
	Feeder.Alarms.xTrayEmptyL2 := Feeder.Inputs.xTrayEmptyL2;
	Feeder.Alarms.xMediaLowL2 := Feeder.Inputs.xMediaLowL2;

	IF Feeder.Inputs.xError THEN
		Feeder.Alarms.xError := TRUE;
	END_IF

	tonNotOnline.IN:=NOT Feeder.Inputs.xOnline AND Feeder.Parameters.xLineInAuto;
	tonNotOnline.PT:=T#1s;
	tonNotOnline();
	IF tonNotOnline.Q THEN Feeder.Alarms.xNotOnline := TRUE; END_IF

	//Saving modbus slave status when comms error raises
	IF EDGEPOS (Feeder.Alarms.xCommsError) THEN
		ModSlaveState := Feeder.Status.Comms.ModSlaveState;
		LastError := Feeder.Status.Comms.LastError;
		LastErrorBlockNum := Feeder.Status.Comms.LastErrorBlockNum;
	END_IF

	//Alarms related to comms
	IF Feeder.Status.Comms.xModuleOk THEN
		IF (NOT Feeder.Inputs.Comms.xRemote) AND Feeder.Parameters.xLineInAuto THEN
			Feeder.Alarms.xNotRemote := TRUE;
		END_IF
	END_IF

	//Data write to ancillaries is critical to be updated properly. So just write block is monitored to raise comms alarm
	//Added ancillary first command used to get it ready to check comms also.
	ton_CommsError.IN := NOT Feeder.Status.Comms.xModuleOk AND (NOT Feeder.Orders.xDisableWriteBlock OR Feeder.Commands.xPrepare);
	ton_CommsError.PT := T#500ms;
	ton_CommsError();

	IF ton_CommsError.Q  THEN
		Feeder.Alarms.xCommsError := TRUE;
	END_IF

	//Alarms Summary
	//Critical
	Feeder.Alarms.xCriticalAlarm:=	Feeder.Alarms.xError OR
									Feeder.Alarms.xNotOnline OR
									Feeder.Alarms.xNoPowered OR
									Feeder.Alarms.xNotRemote OR
									Feeder.Alarms.xCommsError;

	//Warning
	Feeder.Alarms.xWarningAlarm	:=	Feeder.Alarms.xTrayEmptyL1 OR
									Feeder.Alarms.xMediaLowL1 OR
									Feeder.Alarms.xTrayEmptyL2 OR
									Feeder.Alarms.xMediaLowL2;

END_ACTION

ACTION ResetAlarms:
	Feeder.Alarms := AlarmsReseted;
END_ACTION
```

#### Configuration.st
```iecst
ACTION Configuration:

	CASE Feeder.Status.FeederType OF
		FEEDERTY_BOTTOM_14:
			Feeder.Parameters.Hw.iMaxMediaWidth := 1400;
			Feeder.Parameters.Hw.iMaxMediaLength := 3000;
			Feeder.Parameters.Hw.iMinMediaThickness := 8;
			Feeder.Parameters.Hw.iMaxMediaThickness := 160;
			Feeder.Parameters.Hw.xOffsetAvailable := FALSE;
			Feeder.Parameters.Hw.xDoubleLineAllowed := FALSE;

		FEEDERTY_BOTTOM_18:
			Feeder.Parameters.Hw.iMaxMediaWidth := 1800;
			Feeder.Parameters.Hw.iMaxMediaLength := 3000;
			Feeder.Parameters.Hw.iMinMediaThickness := 8;
			Feeder.Parameters.Hw.iMaxMediaThickness := 160;
			Feeder.Parameters.Hw.xOffsetAvailable := TRUE;
			Feeder.Parameters.Hw.iMaxOffset := 15;
			Feeder.Parameters.Hw.iMinOffset := -15;
			Feeder.Parameters.Hw.xDoubleLineAllowed := TRUE;

		FEEDERTY_TOP:
			Feeder.Parameters.Hw.iMaxMediaWidth := 1800;
			Feeder.Parameters.Hw.iMaxMediaLength := 3200;
			Feeder.Parameters.Hw.iMinMediaThickness := 2;
			Feeder.Parameters.Hw.iMaxMediaThickness := 350;
			Feeder.Parameters.Hw.xOffsetAvailable := FALSE;
			Feeder.Parameters.Hw.xDoubleLineAllowed := TRUE;

	END_CASE

END_ACTION
```

#### Feeder.st
```iecst
PROGRAM _CYCLIC

	Feeder ACCESS ADR(gFeeder);

	//Version
	Feeder.Status.Version.iVersion0 := Feeder.Inputs.Comms.iVersion1;
	Feeder.Status.Version.iVersion1 := Feeder.Inputs.Comms.iVersion2;
	Feeder.Status.Version.iVersion2 := Feeder.Inputs.Comms.iVersion3;
	Feeder.Status.Version.iVersion3 := Feeder.Inputs.Comms.iVersion4;

	//Model evaluation
	iFeederModel.0 := Feeder.Inputs.xModelInput[0];
	iFeederModel.1 := Feeder.Inputs.xModelInput[1];
	iFeederModel.2 := Feeder.Inputs.xModelInput[2];

	Feeder.Parameters.xInstalled := iFeederModel>0;

	//Specify Type of Feeder Model
	Feeder.Status.iModel := iFeederModel;
	CASE iFeederModel OF
		1: Feeder.Status.FeederType := FEEDERTY_BOTTOM_14;
		2: Feeder.Status.FeederType := FEEDERTY_BOTTOM_18;
		3: Feeder.Status.FeederType := FEEDERTY_TOP;
		ELSE Feeder.Status.FeederType := FEEDERTY_UNDEFINED;
	END_CASE

	IF NOT Feeder.Parameters.xInstalled OR NOT Feeder.ParSw.xEnabled THEN
		ResetAlarms;
		Feeder.Outputs := OutputsReset;
		Feeder.Commands:=ResetCommands;
		Feeder.Status.DeviceStatus:=FEEDER_TURNED_OFF;
		CopyOfWriteData := EraseWriteData;
		UpdateStatus;
		RETURN;
	END_IF

	IF Feeder.Commands.xResetAlarms THEN ResetAlarms; END_IF

	Configuration;

	Status;

	IF NOT Feeder.Parameters.xSimulationMode THEN
		AssignDataComms;
	END_IF

	//Erasing data when ancillary not in remote
	IF NOT Feeder.Inputs.Comms.xRemote THEN
		CopyOfWriteData := EraseWriteData;
	END_IF

	Alarms;

	IF Feeder.Status.Device.xFaulted OR Feeder.Status.Device.xTurnedOff OR NOT Feeder.Parameters.xLineInAuto THEN
		Feeder.Status.CtrlStatus:=FEEDERCTRL_STOPPED;
	END_IF

	CASE Feeder.Status.CtrlStatus OF
		FEEDERCTRL_STOPPED:
			Feeder.Outputs.Physical := PhysicalOutputsReset;
			IF Feeder.Status.DeviceStatus=FEEDER_INIT AND Feeder.Commands.xPrepare THEN
				Feeder.Status.CtrlStatus:=FEEDERCTRL_PREPARING;
			END_IF

		FEEDERCTRL_STOPPING:
			//Actions
			Feeder.Outputs.Physical := PhysicalOutputsReset;

			//Transition
			IF Feeder.Status.DeviceStatus=FEEDER_TURNED_OFF OR Feeder.Status.DeviceStatus=FEEDER_INIT OR Feeder.Status.DeviceStatus=FEEDER_READY THEN
				Feeder.Status.CtrlStatus:=FEEDERCTRL_STOPPED;
			END_IF

		FEEDERCTRL_CONTROLSTOPPING:

		FEEDERCTRL_PREPARING:
			Feeder.Outputs.Physical.xPrepareToFeed:=TRUE;
			IF Feeder.Status.DeviceStatus=FEEDER_READY THEN
				Feeder.Status.CtrlStatus:=FEEDERCTRL_PREPARED;
			END_IF

		FEEDERCTRL_PAUSED,
		FEEDERCTRL_PREPARED:
			IF Feeder.Commands.xStart THEN
				Feeder.Status.CtrlStatus:=FEEDERCTRL_STARTING;
			END_IF

		FEEDERCTRL_STARTING:
			//Actions
			Feeder.Outputs.Physical.xStartFeeding:=TRUE;

			//Transition
			IF Feeder.Status.DeviceStatus=FEEDER_FEEDING THEN
				Feeder.Status.CtrlStatus:=FEEDERCTRL_FEEDING;
			END_IF

			//Transition
			IF Feeder.Commands.xPause THEN
				Feeder.Status.CtrlStatus:=FEEDERCTRL_PAUSING;
			END_IF

		FEEDERCTRL_FEEDING:
			IF Feeder.Commands.xPause THEN
				Feeder.Status.CtrlStatus:=FEEDERCTRL_PAUSING;
			END_IF

		FEEDERCTRL_PAUSING:
			Feeder.Outputs.Physical.xStartFeeding:=FALSE;
			//Transition
			IF Feeder.Status.DeviceStatus=FEEDER_READY THEN
				Feeder.Status.CtrlStatus:=FEEDERCTRL_PAUSED;
			END_IF

	END_CASE

	IF Feeder.Commands.xStop THEN
		Feeder.Status.CtrlStatus:=FEEDERCTRL_STOPPING;
	ELSIF Feeder.Commands.xControlStop THEN
		Feeder.Status.CtrlStatus:=FEEDERCTRL_CONTROLSTOPPING;
	END_IF

	//Store the history of the status to easy the debug
	IF Feeder.Status.CtrlStatus<>StateHistory[0] THEN
		FOR iIndexHistory:=iHistoryLines TO 1 BY -1 DO
			StateHistory[iIndexHistory]:=StateHistory[iIndexHistory-1];
		END_FOR;
		StateHistory[0]:=Feeder.Status.CtrlStatus;
	END_IF

	Feeder.Commands:=ResetCommands;

END_PROGRAM
```

#### Status.st
```iecst
ACTION Status:

	CASE Feeder.Status.DeviceStatus OF
		FEEDER_TURNED_OFF:
			IF Feeder.Inputs.xFeederPresent AND Feeder.Inputs.xOnline THEN
				Feeder.Status.DeviceStatus:=FEEDER_INIT;
			END_IF

		FEEDER_INIT:
			IF Feeder.Outputs.Physical.xPrepareToFeed THEN
				Feeder.Status.DeviceStatus:=FEEDER_PREPARING;
			END_IF

		FEEDER_PREPARING:
			IF Feeder.Inputs.xReadyToFeed THEN
				Feeder.Status.DeviceStatus:=FEEDER_READY;
			ELSIF NOT Feeder.Outputs.Physical.xPrepareToFeed THEN
				Feeder.Status.DeviceStatus:=FEEDER_INIT;
			END_IF

		FEEDER_READY:
			IF Feeder.Inputs.xFeeding THEN
				Feeder.Status.DeviceStatus:=FEEDER_FEEDING;
			ELSIF NOT Feeder.Inputs.xReadyToFeed THEN
				Feeder.Status.DeviceStatus:=FEEDER_INIT;
			END_IF

		FEEDER_FEEDING:
			IF NOT Feeder.Inputs.xFeeding THEN
				Feeder.Status.DeviceStatus:=FEEDER_INIT;
			END_IF

		FEEDER_FAULTED:
			IF NOT Feeder.Inputs.xError THEN
				Feeder.Status.DeviceStatus:=FEEDER_TURNED_OFF;
			END_IF

	END_CASE

	IF NOT Feeder.Inputs.xFeederPresent THEN
		Feeder.Status.DeviceStatus:=FEEDER_TURNED_OFF;
	END_IF
	IF Feeder.Status.DeviceStatus <> FEEDER_TURNED_OFF AND Feeder.Inputs.xError THEN
		Feeder.Status.DeviceStatus:=FEEDER_FAULTED;
	END_IF

	UpdateStatus;

END_ACTION

ACTION UpdateStatus:

	Feeder.Status.Device.xTurnedOff 	:=	Feeder.Status.DeviceStatus=FEEDER_TURNED_OFF;
	Feeder.Status.Device.xInit 			:=	Feeder.Status.DeviceStatus=FEEDER_INIT;
	Feeder.Status.Device.xPreparing 	:=	Feeder.Status.DeviceStatus=FEEDER_PREPARING;
	Feeder.Status.Device.xReadyToFeed	:=	Feeder.Status.DeviceStatus=FEEDER_READY;
	Feeder.Status.Device.xFeeding 		:=	Feeder.Status.DeviceStatus=FEEDER_FEEDING;
	Feeder.Status.Device.xFaulted 		:=	Feeder.Status.DeviceStatus=FEEDER_FAULTED;

END_ACTION
```

### FeederSim.typ
```iecst
TYPE
	FeederSimCommands_typ : 	STRUCT
		CreateError : BOOL;
	END_STRUCT;
	FeederSim_typ : 	STRUCT
		Commands : FeederSimCommands_typ;
	END_STRUCT;
END_TYPE
```

- Primer.graphml (not shown)

### Program Logical/ExtPack/_Ancillaries/PrimerCtrl/PrimerCtrl_v1/PrimerCtrl

#### Alarms.st
```iecst
ACTION Alarms:

	Primer.Alarms.xNoPrimerPresent:= NOT Primer.Inputs.xPrimerPresent;

	//IF NO Primer, define that alarm and exit
	IF Primer.Alarms.xNoPrimerPresent THEN
		ResetAlarms;
		Primer.Alarms.xNoPrimerPresent:=TRUE;
	END_IF

	//Primer No Powered Warning
	IF Primer.Inputs.xNoPowered THEN Primer.Alarms.xNoPowered := TRUE; END_IF

	Primer.Alarms.xCoatingLevelLow:=Primer.Inputs.xCoatingLevelLow;

	IF Primer.Inputs.xError THEN
		Primer.Alarms.xError := TRUE;
	END_IF

	//Saving modbus slave status when comms error raises
	IF EDGEPOS (Primer.Alarms.xCommsError) THEN
		ModSlaveState := Primer.Status.Comms.ModSlaveState;
		LastError := Primer.Status.Comms.LastError;
		LastErrorBlockNum := Primer.Status.Comms.LastErrorBlockNum;
	END_IF

	//Alarms related to comms
	IF Primer.Status.Comms.xModuleOk THEN
		//Remote
		IF NOT Primer.Inputs.Comms.xRemote AND Primer.Parameters.xLineInAuto THEN
			Primer.Alarms.xNotRemote := TRUE;
		END_IF
		//Stop request
		IF Primer.Inputs.Comms.xStopButtonPressed THEN
			Primer.Alarms.xStopRequest := TRUE;
		END_IF
	END_IF

	//Data write to ancillaries is critical to be updated properly. So just write block is monitored to raise comms alarm
	//Added ancillary first command used to get it ready to check comms also.
	//Read function not considered as the only variable critical for line process is to acknowledge "belt empty" status and in case of module nOk
	//timer "tonEmptyBelt" is executed
	ton_CommsError.IN := NOT Primer.Status.Comms.xModuleOk AND (NOT Primer.Orders.xDisableWriteBlock OR Primer.Commands.xPrepare);
	ton_CommsError.PT := T#500ms;
	ton_CommsError();

	IF ton_CommsError.Q  THEN
		Primer.Alarms.xCommsError := TRUE;
	END_IF

	//Alarms Summary
	//Critical
	Primer.Alarms.xCriticalAlarm:= 	Primer.Alarms.xError OR
									Primer.Alarms.xNoPowered OR
									Primer.Alarms.xNotRemote OR
									Primer.Alarms.xStopRequest OR

									Primer.Alarms.xCommsError;

	//Warning
	//Primer.Alarms.xWarningAlarm	:=	;

END_ACTION

ACTION ResetAlarms:
	Primer.Alarms := AlarmsReseted;
END_ACTION
```

#### AssignDataComms.st
```iecst
ACTION AssignDataComms:

	//Active modbus slave diagnosis when ancillary is enabled. This parameter must remain to TRUE from then on.
	//Just would be set to FALSE via UaExpert, to reset historic errors when ancillary is disabled
	Primer.Parameters.xActiveSlaveDiagnosis := TRUE;

	xBoardParametersChanged := 	(Primer.Parameters.Media.rWidth<>rPrevWidth) OR
								(Primer.Parameters.Media.rLength<>rPrevLength) OR
								(Primer.Parameters.Media.rThickness<>rPrevThickness) OR
								(Primer.Parameters.Media.rGap<>rPrevGap);

	rPrevWidth:=Primer.Parameters.Media.rWidth;
	rPrevLength:=Primer.Parameters.Media.rLength;
	rPrevThickness:=Primer.Parameters.Media.rThickness;
	rPrevGap:=Primer.Parameters.Media.rGap;

	tof_BoardParametersChanged.IN:=xBoardParametersChanged;
	tof_BoardParametersChanged.PT:=t#1s;
	tof_BoardParametersChanged();

	IF Primer.Status.PrimerType = PRIMERTY_DMS THEN
		DmsComms;

	ELSE
		DefaultPrimerComms;
	END_IF

	//Disabling writting after some time active. To test
	tonDisableWrittingOfData.IN:= NOT xDisableWriteData;
	tonDisableWrittingOfData.PT:= T#1000ms;
	tonDisableWrittingOfData();

	IF tonDisableWrittingOfData.Q THEN
		xDisableWriteData := TRUE;
	END_IF

	FOR iIndex:=1 TO 25 DO
		IF gToWriteDataModbPrimer[iIndex]<>CopyOfWriteData[iIndex] THEN
			xDisableWriteData := FALSE;
		END_IF
	END_FOR

	Primer.Orders.xDisableWriteBlock := xDisableWriteData;

	//Copying previous data
	CopyOfWriteData := gToWriteDataModbPrimer;

END_ACTION

ACTION DmsComms:

		/////////////////
		//Pre bits treatment
		Primer.Outputs.Comms.iControl.1 := Primer.Commands.xEnteringMedia;
		Primer.Outputs.Comms.iControl.2 := Primer.Commands.xNewBoardParameters:=tof_BoardParametersChanged.Q;
		//Primer.Outputs.Comms.iControl.3 := ;
		Primer.Outputs.Comms.iControl.4 := TRUE; //Primer.Outputs.Comms.xLineAirSupply;
		Primer.Outputs.Comms.iControl.5 := 	Primer.Parameters.LineState = LINE_PREPARING_EMPTYBELT OR
											Primer.Parameters.LineState = LINE_STARTING_EMPTYBELT OR
											Primer.Parameters.LineState = LINE_BELT_EMPTYING;

		Primer.Outputs.Comms.iControl2.13 := FALSE; //Single line:0, Double line: 1
		Primer.Outputs.Comms.iControl2.15 := TRUE; //Edge:0, Center: 1

		//Write Registers
		gToWriteDataModbPrimer[1] := REAL_TO_UINT(Primer.Parameters.Media.rWidth*10);
		gToWriteDataModbPrimer[2] := REAL_TO_UINT(Primer.Parameters.Media.rLength*10);
		gToWriteDataModbPrimer[3] := REAL_TO_UINT(Primer.Parameters.Media.rThickness*10);
		gToWriteDataModbPrimer[4] := REAL_TO_UINT(Primer.Parameters.Media.rGap*10);
		//gToWriteDataModbPrimer[5] := ;
		gToWriteDataModbPrimer[6] := REAL_TO_UINT(Primer.Parameters.rLineAccelRate*60); //150;
		gToWriteDataModbPrimer[7] := REAL_TO_UINT(Primer.Parameters.rLineDecelRate*60); //150;
		gToWriteDataModbPrimer[8] := REAL_TO_UINT(Primer.Parameters.rBeltSpeedSetPoint*100);
		gToWriteDataModbPrimer[9] := Primer.Outputs.Comms.iControl;;
		gToWriteDataModbPrimer[10] := Primer.Outputs.Comms.iControl2;
		(*
		gToWriteDataModbPrimer[11] := ;
		gToWriteDataModbPrimer[12] := ;
		gToWriteDataModbPrimer[13] := ;
		gToWriteDataModbPrimer[14] := ;
		gToWriteDataModbPrimer[15] := ;

		gToWriteDataModbPrimer[16] := ;
		gToWriteDataModbPrimer[17] := ;

		gToWriteDataModbPrimer[18] := ;
		gToWriteDataModbPrimer[19] := ;
		gToWriteDataModbPrimer[20] := ;

		gToWriteDataModbPrimer[21] := ;
		gToWriteDataModbPrimer[22] := ;
		gToWriteDataModbPrimer[23] := ;
		gToWriteDataModbPrimer[24] := ;
		gToWriteDataModbPrimer[25] := ;
		*)

		////////////////
		//Read Registers
		IF Primer.Status.Comms.xModuleOk THEN
			Primer.Inputs.Comms.iStatus := gReceivedDataModbPrimer[1];
			//Primer.Inputs.Comms. := gReceivedDataModbPrimer[2];
			Primer.Inputs.Comms.uiCoaterRollerSpeed := gReceivedDataModbPrimer[3];
			Primer.Inputs.Comms.uiTransportSpeed := gReceivedDataModbPrimer[4];
			(*
			:= gReceivedDataModbPrimer[5];
			:= gReceivedDataModbPrimer[6];
			:= gReceivedDataModbPrimer[7];
			:= gReceivedDataModbPrimer[8];
			:= gReceivedDataModbPrimer[9];
			:= gReceivedDataModbPrimer[10];

			:= gReceivedDataModbPrimer[11];
			:= gReceivedDataModbPrimer[12];
			:= gReceivedDataModbPrimer[13];
			:= gReceivedDataModbPrimer[14];
			:= gReceivedDataModbPrimer[15];
			*)
			Primer.Inputs.Comms.iVersion1 := gReceivedDataModbPrimer[16];
			Primer.Inputs.Comms.iVersion2 := gReceivedDataModbPrimer[17];
			Primer.Inputs.Comms.iVersion3 := gReceivedDataModbPrimer[18];
			Primer.Inputs.Comms.iVersion4 := gReceivedDataModbPrimer[19];
			(*
			:= gReceivedDataModbPrimer[20];
			:= gReceivedDataModbPrimer[21];
			:= gReceivedDataModbPrimer[22];
			:= gReceivedDataModbPrimer[23];
			:= gReceivedDataModbPrimer[24];
			:= gReceivedDataModbPrimer[25];
			*)
	END_IF

		//Post bit treatment
		Primer.Inputs.Comms.xRemote := Primer.Inputs.Comms.iStatus.1;
		Primer.Inputs.Comms.xBeltEmpty := Primer.Inputs.Comms.iStatus.3;
		Primer.Inputs.Comms.xStopButtonPressed := Primer.Inputs.Comms.iStatus.10;

END_ACTION

ACTION DefaultPrimerComms:

		/////////////////
		//Pre bits treatment
		//Primer.Outputs.Comms.iControl.0 := ;
		//Primer.Outputs.Comms.iControl.1 := ;
		Primer.Outputs.Comms.iControl.2 := Primer.Commands.xNewBoardParameters := tof_BoardParametersChanged.Q;
		//Primer.Outputs.Comms.iControl.3 := ;
		//Primer.Outputs.Comms.iControl.4 := Primer.Outputs.Comms.xLineAirSupply;
		Primer.Outputs.Comms.iControl.5 := 	Primer.Parameters.LineState = LINE_PREPARING_EMPTYBELT OR
											Primer.Parameters.LineState = LINE_STARTING_EMPTYBELT OR
											Primer.Parameters.LineState = LINE_BELT_EMPTYING;

		Primer.Outputs.Comms.iControl.6 := Primer.Parameters.xDoubleLine;

		//Write Registers
		gToWriteDataModbPrimer[1] := Primer.Outputs.Comms.iControl;
		gToWriteDataModbPrimer[2] := REAL_TO_UINT(Primer.Parameters.Media.rLength*10);
		gToWriteDataModbPrimer[3] := REAL_TO_UINT(Primer.Parameters.Media.rWidth*10);
		gToWriteDataModbPrimer[4] := REAL_TO_UINT(Primer.Parameters.Media.rThickness*10);
		gToWriteDataModbPrimer[5] := REAL_TO_UINT(Primer.Parameters.Media.rGap*10);
		gToWriteDataModbPrimer[6] := REAL_TO_UINT(Primer.Parameters.rLineAccelRate*60); //150;
		gToWriteDataModbPrimer[7] := REAL_TO_UINT(Primer.Parameters.rLineDecelRate*60); //150;
		gToWriteDataModbPrimer[8] := REAL_TO_UINT(Primer.Parameters.rBeltSpeedSetPoint*10);
		(*gToWriteDataModbPrimer[9] := ;
		gToWriteDataModbPrimer[10] := ;
		gToWriteDataModbPrimer[11] := ;

		gToWriteDataModbPrimer[12] := ;
		gToWriteDataModbPrimer[13] := ;
		gToWriteDataModbPrimer[14] := ;
		gToWriteDataModbPrimer[15] := ;
		gToWriteDataModbPrimer[16] := ;
		gToWriteDataModbPrimer[17] := ;
		gToWriteDataModbPrimer[18] := ;
		gToWriteDataModbPrimer[19] := ;
		gToWriteDataModbPrimer[20] := ;
		gToWriteDataModbPrimer[21] := ;
		gToWriteDataModbPrimer[22] := ;
		gToWriteDataModbPrimer[23] := ;
		gToWriteDataModbPrimer[24] := ;
		gToWriteDataModbPrimer[25] := ;
		*)

		////////////////
		//Read Registers
		IF Primer.Status.Comms.xModuleOk THEN
			Primer.Inputs.Comms.iStatus := gReceivedDataModbPrimer[1];
			//Primer.Inputs.Comms. := gReceivedDataModbPrimer[2];
			Primer.Inputs.Comms.uiCoaterRollerSpeed := gReceivedDataModbPrimer[3];
			Primer.Inputs.Comms.uiTransportSpeed := gReceivedDataModbPrimer[4];
			(*
			:= gReceivedDataModbPrimer[5];
			:= gReceivedDataModbPrimer[6];
			:= gReceivedDataModbPrimer[7];
			:= gReceivedDataModbPrimer[8];
			:= gReceivedDataModbPrimer[9];
			:= gReceivedDataModbPrimer[10];

			:= gReceivedDataModbPrimer[11];
			:= gReceivedDataModbPrimer[12];
			:= gReceivedDataModbPrimer[13];
			:= gReceivedDataModbPrimer[14];
			:= gReceivedDataModbPrimer[15];
			*)
			Primer.Inputs.Comms.iVersion1 := gReceivedDataModbPrimer[16];
			Primer.Inputs.Comms.iVersion2 := gReceivedDataModbPrimer[17];
			Primer.Inputs.Comms.iVersion3 := gReceivedDataModbPrimer[18];
			Primer.Inputs.Comms.iVersion4 := gReceivedDataModbPrimer[19];
			(*
			:= gReceivedDataModbPrimer[20];
			:= gReceivedDataModbPrimer[21];
			:= gReceivedDataModbPrimer[22];
			:= gReceivedDataModbPrimer[23];
			:= gReceivedDataModbPrimer[24];
			:= gReceivedDataModbPrimer[25];
			*)
	END_IF

		//Post bit treatment
		Primer.Inputs.Comms.xRemote := Primer.Inputs.Comms.iStatus.8;
		Primer.Inputs.Comms.xBeltEmpty := Primer.Inputs.Comms.iStatus.9;

END_ACTION
```
